MoveL RelTool (p1,3.000000,3.000000,9.000000,\Rx:=0.000000,\Ry:=0),vel1,zoneval,Extruder\WObj:=Workobject_1;
MoveL RelTool (p1,5.000000,3.000000,9.000000,\Rx:=0.000000,\Ry:=-0.000000),vel1,zoneval,Extruder\WObj:=Workobject_1;
MoveL RelTool (p1,7.500000,3.000000,9.000000,\Rx:=0.000000,\Ry:=-0.000000),vel1,zoneval,Extruder\WObj:=Workobject_1;
MoveL RelTool (p1,10.000000,3.000000,9.000000,\Rx:=0.000000,\Ry:=-0.000000),vel1,zoneval,Extruder\WObj:=Workobject_1;
MoveL RelTool (p1,12.500000,3.000000,9.000000,\Rx:=0.000000,\Ry:=-0.000000),vel1,zoneval,Extruder\WObj:=Workobject_1;
MoveL RelTool (p1,15.000000,3.000000,9.000000,\Rx:=0.000000,\Ry:=-0.000000),vel1,zoneval,Extruder\WObj:=Workobject_1;
MoveL RelTool (p1,17.500000,3.000000,9.083964,\Rx:=0.000000,\Ry:=-4.411855),vel1,zoneval,Extruder\WObj:=Workobject_1;
MoveL RelTool (p1,20.000000,3.000000,11.367111,\Rx:=0.000000,\Ry:=-10.154539),vel1,zoneval,Extruder\WObj:=Workobject_1;
MoveL RelTool (p1,22.500000,3.000000,13.528177,\Rx:=0.000000,\Ry:=-7.985654),vel1,zoneval,Extruder\WObj:=Workobject_1;
MoveL RelTool (p1,25.000000,3.000000,15.076143,\Rx:=0.000000,\Ry:=-5.751524),vel1,zoneval,Extruder\WObj:=Workobject_1;
MoveL RelTool (p1,27.500000,3.000000,16.224522,\Rx:=0.000000,\Ry:=-4.442626),vel1,zoneval,Extruder\WObj:=Workobject_1;
MoveL RelTool (p1,30.000000,3.000000,17.115741,\Rx:=0.000000,\Ry:=-3.471339),vel1,zoneval,Extruder\WObj:=Workobject_1;
MoveL RelTool (p1,32.500000,3.000000,17.811501,\Rx:=0.000000,\Ry:=-2.537038),vel1,zoneval,Extruder\WObj:=Workobject_1;
MoveL RelTool (p1,35.000000,3.000000,18.316346,\Rx:=0.000000,\Ry:=-2.278631),vel1,zoneval,Extruder\WObj:=Workobject_1;
MoveL RelTool (p1,37.500000,3.000000,18.667838,\Rx:=0.000000,\Ry:=-1.652509),vel1,zoneval,Extruder\WObj:=Workobject_1;
MoveL RelTool (p1,40.000000,3.000000,18.885153,\Rx:=0.000000,\Ry:=-0.809967),vel1,zoneval,Extruder\WObj:=Workobject_1;
MoveL RelTool (p1,42.500000,3.000000,18.988071,\Rx:=0.000000,\Ry:=-0.131676),vel1,zoneval,Extruder\WObj:=Workobject_1;
MoveL RelTool (p1,45.000000,3.000000,18.928943,\Rx:=0.000000,\Ry:=0.547333),vel1,zoneval,Extruder\WObj:=Workobject_1;
MoveL RelTool (p1,47.500000,3.000000,18.755880,\Rx:=0.000000,\Ry:=1.375675),vel1,zoneval,Extruder\WObj:=Workobject_1;
MoveL RelTool (p1,50.000000,3.000000,18.449475,\Rx:=0.000000,\Ry:=2.217990),vel1,zoneval,Extruder\WObj:=Workobject_1;
MoveL RelTool (p1,52.500000,3.000000,17.996328,\Rx:=0.000000,\Ry:=3.108480),vel1,zoneval,Extruder\WObj:=Workobject_1;
MoveL RelTool (p1,55.000000,3.000000,17.373557,\Rx:=0.000000,\Ry:=4.006255),vel1,zoneval,Extruder\WObj:=Workobject_1;
MoveL RelTool (p1,57.500000,3.000000,16.553376,\Rx:=0.000000,\Ry:=5.005887),vel1,zoneval,Extruder\WObj:=Workobject_1;
MoveL RelTool (p1,60.000000,3.000000,15.484711,\Rx:=0.000000,\Ry:=6.061214),vel1,zoneval,Extruder\WObj:=Workobject_1;
MoveL RelTool (p1,62.500000,3.000000,14.090610,\Rx:=0.000000,\Ry:=7.227695),vel1,zoneval,Extruder\WObj:=Workobject_1;
MoveL RelTool (p1,65.000000,3.000000,12.198583,\Rx:=0.000000,\Ry:=9.902860),vel1,zoneval,Extruder\WObj:=Workobject_1;
MoveL RelTool (p1,67.500000,3.000000,9.464073,\Rx:=0.000000,\Ry:=6.326197),vel1,zoneval,Extruder\WObj:=Workobject_1;
MoveL RelTool (p1,70.000000,3.000000,9.000000,\Rx:=0.000000,\Ry:=-0.000000),vel1,zoneval,Extruder\WObj:=Workobject_1;
MoveL RelTool (p1,72.500000,3.000000,9.000000,\Rx:=0.000000,\Ry:=-0.000000),vel1,zoneval,Extruder\WObj:=Workobject_1;
MoveL RelTool (p1,75.000000,3.000000,9.000000,\Rx:=0.000000,\Ry:=-0.000000),vel1,zoneval,Extruder\WObj:=Workobject_1;
MoveL RelTool (p1,77.500000,3.000000,9.000000,\Rx:=0.000000,\Ry:=-0.000000),vel1,zoneval,Extruder\WObj:=Workobject_1;
MoveL RelTool (p1,80.000000,3.000000,9.000000,\Rx:=0.000000,\Ry:=-0.000000),vel1,zoneval,Extruder\WObj:=Workobject_1;
MoveL RelTool (p1,82.500000,3.000000,9.000000,\Rx:=0.000000,\Ry:=-0.000000),vel1,zoneval,Extruder\WObj:=Workobject_1;
MoveL RelTool (p1,80.500000,3.500000,9.000000,\Rx:=0.000000,\Ry:=0.000000),vel1,zoneval,Extruder\WObj:=Workobject_1;
MoveL RelTool (p1,78.000000,3.500000,9.000000,\Rx:=0.000000,\Ry:=0.000000),vel1,zoneval,Extruder\WObj:=Workobject_1;
MoveL RelTool (p1,75.500000,3.500000,9.000000,\Rx:=0.000000,\Ry:=0.000000),vel1,zoneval,Extruder\WObj:=Workobject_1;
MoveL RelTool (p1,73.000000,3.500000,9.000000,\Rx:=0.000000,\Ry:=0.000000),vel1,zoneval,Extruder\WObj:=Workobject_1;
MoveL RelTool (p1,70.500000,3.500000,9.000000,\Rx:=0.000000,\Ry:=0.000000),vel1,zoneval,Extruder\WObj:=Workobject_1;
MoveL RelTool (p1,68.000000,3.500000,9.192958,\Rx:=0.000000,\Ry:=6.326197),vel1,zoneval,Extruder\WObj:=Workobject_1;
MoveL RelTool (p1,65.500000,3.500000,11.706154,\Rx:=0.000000,\Ry:=9.902860),vel1,zoneval,Extruder\WObj:=Workobject_1;
MoveL RelTool (p1,63.000000,3.500000,13.771773,\Rx:=0.000000,\Ry:=7.227695),vel1,zoneval,Extruder\WObj:=Workobject_1;
MoveL RelTool (p1,60.500000,3.500000,15.226913,\Rx:=0.000000,\Ry:=6.061214),vel1,zoneval,Extruder\WObj:=Workobject_1;
MoveL RelTool (p1,58.000000,3.500000,16.345998,\Rx:=0.000000,\Ry:=5.005887),vel1,zoneval,Extruder\WObj:=Workobject_1;
MoveL RelTool (p1,55.500000,3.500000,17.210825,\Rx:=0.000000,\Ry:=4.006255),vel1,zoneval,Extruder\WObj:=Workobject_1;
MoveL RelTool (p1,53.000000,3.500000,17.871774,\Rx:=0.000000,\Ry:=3.108480),vel1,zoneval,Extruder\WObj:=Workobject_1;
MoveL RelTool (p1,50.500000,3.500000,18.361483,\Rx:=0.000000,\Ry:=2.217990),vel1,zoneval,Extruder\WObj:=Workobject_1;
MoveL RelTool (p1,48.000000,3.500000,18.701647,\Rx:=0.000000,\Ry:=1.375675),vel1,zoneval,Extruder\WObj:=Workobject_1;
MoveL RelTool (p1,45.500000,3.500000,18.907436,\Rx:=0.000000,\Ry:=0.547333),vel1,zoneval,Extruder\WObj:=Workobject_1;
MoveL RelTool (p1,43.000000,3.500000,18.993242,\Rx:=0.000000,\Ry:=-0.131676),vel1,zoneval,Extruder\WObj:=Workobject_1;
MoveL RelTool (p1,40.500000,3.500000,18.917003,\Rx:=0.000000,\Ry:=-0.809967),vel1,zoneval,Extruder\WObj:=Workobject_1;
MoveL RelTool (p1,38.000000,3.500000,18.733099,\Rx:=0.000000,\Ry:=-1.652509),vel1,zoneval,Extruder\WObj:=Workobject_1;
MoveL RelTool (p1,35.500000,3.500000,18.406795,\Rx:=0.000000,\Ry:=-2.278631),vel1,zoneval,Extruder\WObj:=Workobject_1;
MoveL RelTool (p1,33.000000,3.500000,17.912470,\Rx:=0.000000,\Ry:=-2.537038),vel1,zoneval,Extruder\WObj:=Workobject_1;
MoveL RelTool (p1,30.500000,3.500000,17.255542,\Rx:=0.000000,\Ry:=-3.471339),vel1,zoneval,Extruder\WObj:=Workobject_1;
MoveL RelTool (p1,28.000000,3.500000,16.406426,\Rx:=0.000000,\Ry:=-4.442626),vel1,zoneval,Extruder\WObj:=Workobject_1;
MoveL RelTool (p1,25.500000,3.500000,15.318735,\Rx:=0.000000,\Ry:=-5.751524),vel1,zoneval,Extruder\WObj:=Workobject_1;
MoveL RelTool (p1,23.000000,3.500000,13.890588,\Rx:=0.000000,\Ry:=-7.985654),vel1,zoneval,Extruder\WObj:=Workobject_1;
MoveL RelTool (p1,20.500000,3.500000,11.879398,\Rx:=0.000000,\Ry:=-10.154539),vel1,zoneval,Extruder\WObj:=Workobject_1;
MoveL RelTool (p1,18.000000,3.500000,9.264501,\Rx:=0.000000,\Ry:=-4.411855),vel1,zoneval,Extruder\WObj:=Workobject_1;
MoveL RelTool (p1,15.500000,3.500000,9.000000,\Rx:=0.000000,\Ry:=0.000000),vel1,zoneval,Extruder\WObj:=Workobject_1;
MoveL RelTool (p1,13.000000,3.500000,9.000000,\Rx:=0.000000,\Ry:=0.000000),vel1,zoneval,Extruder\WObj:=Workobject_1;
MoveL RelTool (p1,10.500000,3.500000,9.000000,\Rx:=0.000000,\Ry:=0.000000),vel1,zoneval,Extruder\WObj:=Workobject_1;
MoveL RelTool (p1,8.000000,3.500000,9.000000,\Rx:=0.000000,\Ry:=0.000000),vel1,zoneval,Extruder\WObj:=Workobject_1;
MoveL RelTool (p1,5.500000,3.500000,9.000000,\Rx:=0.000000,\Ry:=0.000000),vel1,zoneval,Extruder\WObj:=Workobject_1;
MoveL RelTool (p1,3.000000,3.500000,9.000000,\Rx:=0.000000,\Ry:=0.000000),vel1,zoneval,Extruder\WObj:=Workobject_1;
MoveL RelTool (p1,5.000000,4.000000,9.000000,\Rx:=0.000000,\Ry:=-0.000000),vel1,zoneval,Extruder\WObj:=Workobject_1;
MoveL RelTool (p1,7.500000,4.000000,9.000000,\Rx:=0.000000,\Ry:=-0.000000),vel1,zoneval,Extruder\WObj:=Workobject_1;
MoveL RelTool (p1,10.000000,4.000000,9.000000,\Rx:=0.000000,\Ry:=-0.000000),vel1,zoneval,Extruder\WObj:=Workobject_1;
MoveL RelTool (p1,12.500000,4.000000,9.000000,\Rx:=0.000000,\Ry:=-0.000000),vel1,zoneval,Extruder\WObj:=Workobject_1;
MoveL RelTool (p1,15.000000,4.000000,9.000000,\Rx:=0.000000,\Ry:=-0.000000),vel1,zoneval,Extruder\WObj:=Workobject_1;
MoveL RelTool (p1,17.500000,4.000000,9.083964,\Rx:=0.000000,\Ry:=-4.411855),vel1,zoneval,Extruder\WObj:=Workobject_1;
MoveL RelTool (p1,20.000000,4.000000,11.367111,\Rx:=0.000000,\Ry:=-10.154539),vel1,zoneval,Extruder\WObj:=Workobject_1;
MoveL RelTool (p1,22.500000,4.000000,13.528177,\Rx:=0.000000,\Ry:=-7.985654),vel1,zoneval,Extruder\WObj:=Workobject_1;
MoveL RelTool (p1,25.000000,4.000000,15.076143,\Rx:=0.000000,\Ry:=-5.751524),vel1,zoneval,Extruder\WObj:=Workobject_1;
MoveL RelTool (p1,27.500000,4.000000,16.224522,\Rx:=0.000000,\Ry:=-4.442626),vel1,zoneval,Extruder\WObj:=Workobject_1;
MoveL RelTool (p1,30.000000,4.000000,17.115741,\Rx:=0.000000,\Ry:=-3.471339),vel1,zoneval,Extruder\WObj:=Workobject_1;
MoveL RelTool (p1,32.500000,4.000000,17.811501,\Rx:=0.000000,\Ry:=-2.537038),vel1,zoneval,Extruder\WObj:=Workobject_1;
MoveL RelTool (p1,35.000000,4.000000,18.316346,\Rx:=0.000000,\Ry:=-2.278631),vel1,zoneval,Extruder\WObj:=Workobject_1;
MoveL RelTool (p1,37.500000,4.000000,18.667838,\Rx:=0.000000,\Ry:=-1.652509),vel1,zoneval,Extruder\WObj:=Workobject_1;
MoveL RelTool (p1,40.000000,4.000000,18.885153,\Rx:=0.000000,\Ry:=-0.809967),vel1,zoneval,Extruder\WObj:=Workobject_1;
MoveL RelTool (p1,42.500000,4.000000,18.988071,\Rx:=0.000000,\Ry:=-0.131676),vel1,zoneval,Extruder\WObj:=Workobject_1;
MoveL RelTool (p1,45.000000,4.000000,18.928943,\Rx:=0.000000,\Ry:=0.547333),vel1,zoneval,Extruder\WObj:=Workobject_1;
MoveL RelTool (p1,47.500000,4.000000,18.755880,\Rx:=0.000000,\Ry:=1.375675),vel1,zoneval,Extruder\WObj:=Workobject_1;
MoveL RelTool (p1,50.000000,4.000000,18.449475,\Rx:=0.000000,\Ry:=2.217990),vel1,zoneval,Extruder\WObj:=Workobject_1;
MoveL RelTool (p1,52.500000,4.000000,17.996328,\Rx:=0.000000,\Ry:=3.108480),vel1,zoneval,Extruder\WObj:=Workobject_1;
MoveL RelTool (p1,55.000000,4.000000,17.373557,\Rx:=0.000000,\Ry:=4.006255),vel1,zoneval,Extruder\WObj:=Workobject_1;
MoveL RelTool (p1,57.500000,4.000000,16.553376,\Rx:=0.000000,\Ry:=5.005887),vel1,zoneval,Extruder\WObj:=Workobject_1;
MoveL RelTool (p1,60.000000,4.000000,15.484711,\Rx:=0.000000,\Ry:=6.061214),vel1,zoneval,Extruder\WObj:=Workobject_1;
MoveL RelTool (p1,62.500000,4.000000,14.090610,\Rx:=0.000000,\Ry:=7.227695),vel1,zoneval,Extruder\WObj:=Workobject_1;
MoveL RelTool (p1,65.000000,4.000000,12.198583,\Rx:=0.000000,\Ry:=9.902860),vel1,zoneval,Extruder\WObj:=Workobject_1;
MoveL RelTool (p1,67.500000,4.000000,9.464073,\Rx:=0.000000,\Ry:=6.326197),vel1,zoneval,Extruder\WObj:=Workobject_1;
MoveL RelTool (p1,70.000000,4.000000,9.000000,\Rx:=0.000000,\Ry:=-0.000000),vel1,zoneval,Extruder\WObj:=Workobject_1;
MoveL RelTool (p1,72.500000,4.000000,9.000000,\Rx:=0.000000,\Ry:=-0.000000),vel1,zoneval,Extruder\WObj:=Workobject_1;
MoveL RelTool (p1,75.000000,4.000000,9.000000,\Rx:=0.000000,\Ry:=-0.000000),vel1,zoneval,Extruder\WObj:=Workobject_1;
MoveL RelTool (p1,77.500000,4.000000,9.000000,\Rx:=0.000000,\Ry:=-0.000000),vel1,zoneval,Extruder\WObj:=Workobject_1;
MoveL RelTool (p1,80.000000,4.000000,9.000000,\Rx:=0.000000,\Ry:=-0.000000),vel1,zoneval,Extruder\WObj:=Workobject_1;
MoveL RelTool (p1,82.500000,4.000000,9.000000,\Rx:=0.000000,\Ry:=-0.000000),vel1,zoneval,Extruder\WObj:=Workobject_1;
MoveL RelTool (p1,80.500000,4.500000,9.000000,\Rx:=0.000000,\Ry:=0.000000),vel1,zoneval,Extruder\WObj:=Workobject_1;
MoveL RelTool (p1,78.000000,4.500000,9.000000,\Rx:=0.000000,\Ry:=0.000000),vel1,zoneval,Extruder\WObj:=Workobject_1;
MoveL RelTool (p1,75.500000,4.500000,9.000000,\Rx:=0.000000,\Ry:=0.000000),vel1,zoneval,Extruder\WObj:=Workobject_1;
MoveL RelTool (p1,73.000000,4.500000,9.000000,\Rx:=0.000000,\Ry:=0.000000),vel1,zoneval,Extruder\WObj:=Workobject_1;
MoveL RelTool (p1,70.500000,4.500000,9.000000,\Rx:=0.000000,\Ry:=0.000000),vel1,zoneval,Extruder\WObj:=Workobject_1;
MoveL RelTool (p1,68.000000,4.500000,9.192958,\Rx:=0.000000,\Ry:=6.326197),vel1,zoneval,Extruder\WObj:=Workobject_1;
MoveL RelTool (p1,65.500000,4.500000,11.706154,\Rx:=0.000000,\Ry:=9.902860),vel1,zoneval,Extruder\WObj:=Workobject_1;
MoveL RelTool (p1,63.000000,4.500000,13.771773,\Rx:=0.000000,\Ry:=7.227695),vel1,zoneval,Extruder\WObj:=Workobject_1;
MoveL RelTool (p1,60.500000,4.500000,15.226913,\Rx:=0.000000,\Ry:=6.061214),vel1,zoneval,Extruder\WObj:=Workobject_1;
MoveL RelTool (p1,58.000000,4.500000,16.345998,\Rx:=0.000000,\Ry:=5.005887),vel1,zoneval,Extruder\WObj:=Workobject_1;
MoveL RelTool (p1,55.500000,4.500000,17.210825,\Rx:=0.000000,\Ry:=4.006255),vel1,zoneval,Extruder\WObj:=Workobject_1;
MoveL RelTool (p1,53.000000,4.500000,17.871774,\Rx:=0.000000,\Ry:=3.108480),vel1,zoneval,Extruder\WObj:=Workobject_1;
MoveL RelTool (p1,50.500000,4.500000,18.361483,\Rx:=0.000000,\Ry:=2.217990),vel1,zoneval,Extruder\WObj:=Workobject_1;
MoveL RelTool (p1,48.000000,4.500000,18.701647,\Rx:=0.000000,\Ry:=1.375675),vel1,zoneval,Extruder\WObj:=Workobject_1;
MoveL RelTool (p1,45.500000,4.500000,18.907436,\Rx:=0.000000,\Ry:=0.547333),vel1,zoneval,Extruder\WObj:=Workobject_1;
MoveL RelTool (p1,43.000000,4.500000,18.993242,\Rx:=0.000000,\Ry:=-0.131676),vel1,zoneval,Extruder\WObj:=Workobject_1;
MoveL RelTool (p1,40.500000,4.500000,18.917003,\Rx:=0.000000,\Ry:=-0.809967),vel1,zoneval,Extruder\WObj:=Workobject_1;
MoveL RelTool (p1,38.000000,4.500000,18.733099,\Rx:=0.000000,\Ry:=-1.652509),vel1,zoneval,Extruder\WObj:=Workobject_1;
MoveL RelTool (p1,35.500000,4.500000,18.406795,\Rx:=0.000000,\Ry:=-2.278631),vel1,zoneval,Extruder\WObj:=Workobject_1;
MoveL RelTool (p1,33.000000,4.500000,17.912470,\Rx:=0.000000,\Ry:=-2.537038),vel1,zoneval,Extruder\WObj:=Workobject_1;
MoveL RelTool (p1,30.500000,4.500000,17.255542,\Rx:=0.000000,\Ry:=-3.471339),vel1,zoneval,Extruder\WObj:=Workobject_1;
MoveL RelTool (p1,28.000000,4.500000,16.406426,\Rx:=0.000000,\Ry:=-4.442626),vel1,zoneval,Extruder\WObj:=Workobject_1;
MoveL RelTool (p1,25.500000,4.500000,15.318735,\Rx:=0.000000,\Ry:=-5.751524),vel1,zoneval,Extruder\WObj:=Workobject_1;
MoveL RelTool (p1,23.000000,4.500000,13.890588,\Rx:=0.000000,\Ry:=-7.985654),vel1,zoneval,Extruder\WObj:=Workobject_1;
MoveL RelTool (p1,20.500000,4.500000,11.879398,\Rx:=0.000000,\Ry:=-10.154539),vel1,zoneval,Extruder\WObj:=Workobject_1;
MoveL RelTool (p1,18.000000,4.500000,9.264501,\Rx:=0.000000,\Ry:=-4.411855),vel1,zoneval,Extruder\WObj:=Workobject_1;
MoveL RelTool (p1,15.500000,4.500000,9.000000,\Rx:=0.000000,\Ry:=0.000000),vel1,zoneval,Extruder\WObj:=Workobject_1;
MoveL RelTool (p1,13.000000,4.500000,9.000000,\Rx:=0.000000,\Ry:=0.000000),vel1,zoneval,Extruder\WObj:=Workobject_1;
MoveL RelTool (p1,10.500000,4.500000,9.000000,\Rx:=0.000000,\Ry:=0.000000),vel1,zoneval,Extruder\WObj:=Workobject_1;
MoveL RelTool (p1,8.000000,4.500000,9.000000,\Rx:=0.000000,\Ry:=0.000000),vel1,zoneval,Extruder\WObj:=Workobject_1;
MoveL RelTool (p1,5.500000,4.500000,9.000000,\Rx:=0.000000,\Ry:=0.000000),vel1,zoneval,Extruder\WObj:=Workobject_1;
MoveL RelTool (p1,3.000000,4.500000,9.000000,\Rx:=0.000000,\Ry:=0.000000),vel1,zoneval,Extruder\WObj:=Workobject_1;
MoveL RelTool (p1,5.000000,5.000000,9.000000,\Rx:=0.000000,\Ry:=-0.000000),vel1,zoneval,Extruder\WObj:=Workobject_1;
MoveL RelTool (p1,7.500000,5.000000,9.000000,\Rx:=0.000000,\Ry:=-0.000000),vel1,zoneval,Extruder\WObj:=Workobject_1;
MoveL RelTool (p1,10.000000,5.000000,9.000000,\Rx:=0.000000,\Ry:=-0.000000),vel1,zoneval,Extruder\WObj:=Workobject_1;
MoveL RelTool (p1,12.500000,5.000000,9.000000,\Rx:=0.000000,\Ry:=-0.000000),vel1,zoneval,Extruder\WObj:=Workobject_1;
MoveL RelTool (p1,15.000000,5.000000,9.000000,\Rx:=0.000000,\Ry:=-0.000000),vel1,zoneval,Extruder\WObj:=Workobject_1;
MoveL RelTool (p1,17.500000,5.000000,9.083964,\Rx:=0.000000,\Ry:=-4.411855),vel1,zoneval,Extruder\WObj:=Workobject_1;
MoveL RelTool (p1,20.000000,5.000000,11.367111,\Rx:=0.000000,\Ry:=-10.154539),vel1,zoneval,Extruder\WObj:=Workobject_1;
MoveL RelTool (p1,22.500000,5.000000,13.528177,\Rx:=0.000000,\Ry:=-7.985654),vel1,zoneval,Extruder\WObj:=Workobject_1;
MoveL RelTool (p1,25.000000,5.000000,15.076143,\Rx:=0.000000,\Ry:=-5.751524),vel1,zoneval,Extruder\WObj:=Workobject_1;
MoveL RelTool (p1,27.500000,5.000000,16.224522,\Rx:=0.000000,\Ry:=-4.442626),vel1,zoneval,Extruder\WObj:=Workobject_1;
MoveL RelTool (p1,30.000000,5.000000,17.115741,\Rx:=0.000000,\Ry:=-3.471339),vel1,zoneval,Extruder\WObj:=Workobject_1;
MoveL RelTool (p1,32.500000,5.000000,17.811501,\Rx:=0.000000,\Ry:=-2.537038),vel1,zoneval,Extruder\WObj:=Workobject_1;
MoveL RelTool (p1,35.000000,5.000000,18.316346,\Rx:=0.000000,\Ry:=-2.278631),vel1,zoneval,Extruder\WObj:=Workobject_1;
MoveL RelTool (p1,37.500000,5.000000,18.667838,\Rx:=0.000000,\Ry:=-1.652509),vel1,zoneval,Extruder\WObj:=Workobject_1;
MoveL RelTool (p1,40.000000,5.000000,18.885153,\Rx:=0.000000,\Ry:=-0.809967),vel1,zoneval,Extruder\WObj:=Workobject_1;
MoveL RelTool (p1,42.500000,5.000000,18.988071,\Rx:=0.000000,\Ry:=-0.131676),vel1,zoneval,Extruder\WObj:=Workobject_1;
MoveL RelTool (p1,45.000000,5.000000,18.928943,\Rx:=0.000000,\Ry:=0.547333),vel1,zoneval,Extruder\WObj:=Workobject_1;
MoveL RelTool (p1,47.500000,5.000000,18.755880,\Rx:=0.000000,\Ry:=1.375675),vel1,zoneval,Extruder\WObj:=Workobject_1;
MoveL RelTool (p1,50.000000,5.000000,18.449475,\Rx:=0.000000,\Ry:=2.217990),vel1,zoneval,Extruder\WObj:=Workobject_1;
MoveL RelTool (p1,52.500000,5.000000,17.996328,\Rx:=0.000000,\Ry:=3.108480),vel1,zoneval,Extruder\WObj:=Workobject_1;
MoveL RelTool (p1,55.000000,5.000000,17.373557,\Rx:=0.000000,\Ry:=4.006255),vel1,zoneval,Extruder\WObj:=Workobject_1;
MoveL RelTool (p1,57.500000,5.000000,16.553376,\Rx:=0.000000,\Ry:=5.005887),vel1,zoneval,Extruder\WObj:=Workobject_1;
MoveL RelTool (p1,60.000000,5.000000,15.484711,\Rx:=0.000000,\Ry:=6.061214),vel1,zoneval,Extruder\WObj:=Workobject_1;
MoveL RelTool (p1,62.500000,5.000000,14.090610,\Rx:=0.000000,\Ry:=7.227695),vel1,zoneval,Extruder\WObj:=Workobject_1;
MoveL RelTool (p1,65.000000,5.000000,12.198583,\Rx:=0.000000,\Ry:=9.902860),vel1,zoneval,Extruder\WObj:=Workobject_1;
MoveL RelTool (p1,67.500000,5.000000,9.464073,\Rx:=0.000000,\Ry:=6.326197),vel1,zoneval,Extruder\WObj:=Workobject_1;
MoveL RelTool (p1,70.000000,5.000000,9.000000,\Rx:=0.000000,\Ry:=-0.000000),vel1,zoneval,Extruder\WObj:=Workobject_1;
MoveL RelTool (p1,72.500000,5.000000,9.000000,\Rx:=0.000000,\Ry:=-0.000000),vel1,zoneval,Extruder\WObj:=Workobject_1;
MoveL RelTool (p1,75.000000,5.000000,9.000000,\Rx:=0.000000,\Ry:=-0.000000),vel1,zoneval,Extruder\WObj:=Workobject_1;
MoveL RelTool (p1,77.500000,5.000000,9.000000,\Rx:=0.000000,\Ry:=-0.000000),vel1,zoneval,Extruder\WObj:=Workobject_1;
MoveL RelTool (p1,80.000000,5.000000,9.000000,\Rx:=0.000000,\Ry:=-0.000000),vel1,zoneval,Extruder\WObj:=Workobject_1;
MoveL RelTool (p1,82.500000,5.000000,9.000000,\Rx:=0.000000,\Ry:=-0.000000),vel1,zoneval,Extruder\WObj:=Workobject_1;
MoveL RelTool (p1,80.500000,5.500000,9.000000,\Rx:=0.000000,\Ry:=0.000000),vel1,zoneval,Extruder\WObj:=Workobject_1;
MoveL RelTool (p1,78.000000,5.500000,9.000000,\Rx:=0.000000,\Ry:=0.000000),vel1,zoneval,Extruder\WObj:=Workobject_1;
MoveL RelTool (p1,75.500000,5.500000,9.000000,\Rx:=0.000000,\Ry:=0.000000),vel1,zoneval,Extruder\WObj:=Workobject_1;
MoveL RelTool (p1,73.000000,5.500000,9.000000,\Rx:=0.000000,\Ry:=0.000000),vel1,zoneval,Extruder\WObj:=Workobject_1;
MoveL RelTool (p1,70.500000,5.500000,9.000000,\Rx:=0.000000,\Ry:=0.000000),vel1,zoneval,Extruder\WObj:=Workobject_1;
MoveL RelTool (p1,68.000000,5.500000,9.192958,\Rx:=0.000000,\Ry:=6.326197),vel1,zoneval,Extruder\WObj:=Workobject_1;
MoveL RelTool (p1,65.500000,5.500000,11.706154,\Rx:=0.000000,\Ry:=9.902860),vel1,zoneval,Extruder\WObj:=Workobject_1;
MoveL RelTool (p1,63.000000,5.500000,13.771773,\Rx:=0.000000,\Ry:=7.227695),vel1,zoneval,Extruder\WObj:=Workobject_1;
MoveL RelTool (p1,60.500000,5.500000,15.226913,\Rx:=0.000000,\Ry:=6.061214),vel1,zoneval,Extruder\WObj:=Workobject_1;
MoveL RelTool (p1,58.000000,5.500000,16.345998,\Rx:=0.000000,\Ry:=5.005887),vel1,zoneval,Extruder\WObj:=Workobject_1;
MoveL RelTool (p1,55.500000,5.500000,17.210825,\Rx:=0.000000,\Ry:=4.006255),vel1,zoneval,Extruder\WObj:=Workobject_1;
MoveL RelTool (p1,53.000000,5.500000,17.871774,\Rx:=0.000000,\Ry:=3.108480),vel1,zoneval,Extruder\WObj:=Workobject_1;
MoveL RelTool (p1,50.500000,5.500000,18.361483,\Rx:=0.000000,\Ry:=2.217990),vel1,zoneval,Extruder\WObj:=Workobject_1;
MoveL RelTool (p1,48.000000,5.500000,18.701647,\Rx:=0.000000,\Ry:=1.375675),vel1,zoneval,Extruder\WObj:=Workobject_1;
MoveL RelTool (p1,45.500000,5.500000,18.907436,\Rx:=0.000000,\Ry:=0.547333),vel1,zoneval,Extruder\WObj:=Workobject_1;
MoveL RelTool (p1,43.000000,5.500000,18.993242,\Rx:=0.000000,\Ry:=-0.131676),vel1,zoneval,Extruder\WObj:=Workobject_1;
MoveL RelTool (p1,40.500000,5.500000,18.917003,\Rx:=0.000000,\Ry:=-0.809967),vel1,zoneval,Extruder\WObj:=Workobject_1;
MoveL RelTool (p1,38.000000,5.500000,18.733099,\Rx:=0.000000,\Ry:=-1.652509),vel1,zoneval,Extruder\WObj:=Workobject_1;
MoveL RelTool (p1,35.500000,5.500000,18.406795,\Rx:=0.000000,\Ry:=-2.278631),vel1,zoneval,Extruder\WObj:=Workobject_1;
MoveL RelTool (p1,33.000000,5.500000,17.912470,\Rx:=0.000000,\Ry:=-2.537038),vel1,zoneval,Extruder\WObj:=Workobject_1;
MoveL RelTool (p1,30.500000,5.500000,17.255542,\Rx:=0.000000,\Ry:=-3.471339),vel1,zoneval,Extruder\WObj:=Workobject_1;
MoveL RelTool (p1,28.000000,5.500000,16.406426,\Rx:=0.000000,\Ry:=-4.442626),vel1,zoneval,Extruder\WObj:=Workobject_1;
MoveL RelTool (p1,25.500000,5.500000,15.318735,\Rx:=0.000000,\Ry:=-5.751524),vel1,zoneval,Extruder\WObj:=Workobject_1;
MoveL RelTool (p1,23.000000,5.500000,13.890588,\Rx:=0.000000,\Ry:=-7.985654),vel1,zoneval,Extruder\WObj:=Workobject_1;
MoveL RelTool (p1,20.500000,5.500000,11.879398,\Rx:=0.000000,\Ry:=-10.154539),vel1,zoneval,Extruder\WObj:=Workobject_1;
MoveL RelTool (p1,18.000000,5.500000,9.264501,\Rx:=0.000000,\Ry:=-4.411855),vel1,zoneval,Extruder\WObj:=Workobject_1;
MoveL RelTool (p1,15.500000,5.500000,9.000000,\Rx:=0.000000,\Ry:=0.000000),vel1,zoneval,Extruder\WObj:=Workobject_1;
MoveL RelTool (p1,13.000000,5.500000,9.000000,\Rx:=0.000000,\Ry:=0.000000),vel1,zoneval,Extruder\WObj:=Workobject_1;
MoveL RelTool (p1,10.500000,5.500000,9.000000,\Rx:=0.000000,\Ry:=0.000000),vel1,zoneval,Extruder\WObj:=Workobject_1;
MoveL RelTool (p1,8.000000,5.500000,9.000000,\Rx:=0.000000,\Ry:=0.000000),vel1,zoneval,Extruder\WObj:=Workobject_1;
MoveL RelTool (p1,5.500000,5.500000,9.000000,\Rx:=0.000000,\Ry:=0.000000),vel1,zoneval,Extruder\WObj:=Workobject_1;
MoveL RelTool (p1,3.000000,5.500000,9.000000,\Rx:=0.000000,\Ry:=0.000000),vel1,zoneval,Extruder\WObj:=Workobject_1;
MoveL RelTool (p1,5.000000,6.000000,9.000000,\Rx:=0.000000,\Ry:=-0.000000),vel1,zoneval,Extruder\WObj:=Workobject_1;
MoveL RelTool (p1,7.500000,6.000000,9.000000,\Rx:=0.000000,\Ry:=-0.000000),vel1,zoneval,Extruder\WObj:=Workobject_1;
MoveL RelTool (p1,10.000000,6.000000,9.000000,\Rx:=0.000000,\Ry:=-0.000000),vel1,zoneval,Extruder\WObj:=Workobject_1;
MoveL RelTool (p1,12.500000,6.000000,9.000000,\Rx:=0.000000,\Ry:=-0.000000),vel1,zoneval,Extruder\WObj:=Workobject_1;
MoveL RelTool (p1,15.000000,6.000000,9.000000,\Rx:=0.000000,\Ry:=-0.000000),vel1,zoneval,Extruder\WObj:=Workobject_1;
MoveL RelTool (p1,17.500000,6.000000,9.083964,\Rx:=0.000000,\Ry:=-4.411855),vel1,zoneval,Extruder\WObj:=Workobject_1;
MoveL RelTool (p1,20.000000,6.000000,11.367111,\Rx:=0.000000,\Ry:=-10.154539),vel1,zoneval,Extruder\WObj:=Workobject_1;
MoveL RelTool (p1,22.500000,6.000000,13.528177,\Rx:=0.000000,\Ry:=-7.985654),vel1,zoneval,Extruder\WObj:=Workobject_1;
MoveL RelTool (p1,25.000000,6.000000,15.076143,\Rx:=0.000000,\Ry:=-5.751524),vel1,zoneval,Extruder\WObj:=Workobject_1;
MoveL RelTool (p1,27.500000,6.000000,16.224522,\Rx:=0.000000,\Ry:=-4.442626),vel1,zoneval,Extruder\WObj:=Workobject_1;
MoveL RelTool (p1,30.000000,6.000000,17.115741,\Rx:=0.000000,\Ry:=-3.471339),vel1,zoneval,Extruder\WObj:=Workobject_1;
MoveL RelTool (p1,32.500000,6.000000,17.811501,\Rx:=0.000000,\Ry:=-2.537038),vel1,zoneval,Extruder\WObj:=Workobject_1;
MoveL RelTool (p1,35.000000,6.000000,18.316346,\Rx:=0.000000,\Ry:=-2.278631),vel1,zoneval,Extruder\WObj:=Workobject_1;
MoveL RelTool (p1,37.500000,6.000000,18.667838,\Rx:=0.000000,\Ry:=-1.652509),vel1,zoneval,Extruder\WObj:=Workobject_1;
MoveL RelTool (p1,40.000000,6.000000,18.885153,\Rx:=0.000000,\Ry:=-0.809967),vel1,zoneval,Extruder\WObj:=Workobject_1;
MoveL RelTool (p1,42.500000,6.000000,18.988071,\Rx:=0.000000,\Ry:=-0.131676),vel1,zoneval,Extruder\WObj:=Workobject_1;
MoveL RelTool (p1,45.000000,6.000000,18.928943,\Rx:=0.000000,\Ry:=0.547333),vel1,zoneval,Extruder\WObj:=Workobject_1;
MoveL RelTool (p1,47.500000,6.000000,18.755880,\Rx:=0.000000,\Ry:=1.375675),vel1,zoneval,Extruder\WObj:=Workobject_1;
MoveL RelTool (p1,50.000000,6.000000,18.449475,\Rx:=0.000000,\Ry:=2.217990),vel1,zoneval,Extruder\WObj:=Workobject_1;
MoveL RelTool (p1,52.500000,6.000000,17.996328,\Rx:=0.000000,\Ry:=3.108480),vel1,zoneval,Extruder\WObj:=Workobject_1;
MoveL RelTool (p1,55.000000,6.000000,17.373557,\Rx:=0.000000,\Ry:=4.006255),vel1,zoneval,Extruder\WObj:=Workobject_1;
MoveL RelTool (p1,57.500000,6.000000,16.553376,\Rx:=0.000000,\Ry:=5.005887),vel1,zoneval,Extruder\WObj:=Workobject_1;
MoveL RelTool (p1,60.000000,6.000000,15.484711,\Rx:=0.000000,\Ry:=6.061214),vel1,zoneval,Extruder\WObj:=Workobject_1;
MoveL RelTool (p1,62.500000,6.000000,14.090610,\Rx:=0.000000,\Ry:=7.227695),vel1,zoneval,Extruder\WObj:=Workobject_1;
MoveL RelTool (p1,65.000000,6.000000,12.198583,\Rx:=0.000000,\Ry:=9.902860),vel1,zoneval,Extruder\WObj:=Workobject_1;
MoveL RelTool (p1,67.500000,6.000000,9.464073,\Rx:=0.000000,\Ry:=6.326197),vel1,zoneval,Extruder\WObj:=Workobject_1;
MoveL RelTool (p1,70.000000,6.000000,9.000000,\Rx:=0.000000,\Ry:=-0.000000),vel1,zoneval,Extruder\WObj:=Workobject_1;
MoveL RelTool (p1,72.500000,6.000000,9.000000,\Rx:=0.000000,\Ry:=-0.000000),vel1,zoneval,Extruder\WObj:=Workobject_1;
MoveL RelTool (p1,75.000000,6.000000,9.000000,\Rx:=0.000000,\Ry:=-0.000000),vel1,zoneval,Extruder\WObj:=Workobject_1;
MoveL RelTool (p1,77.500000,6.000000,9.000000,\Rx:=0.000000,\Ry:=-0.000000),vel1,zoneval,Extruder\WObj:=Workobject_1;
MoveL RelTool (p1,80.000000,6.000000,9.000000,\Rx:=0.000000,\Ry:=-0.000000),vel1,zoneval,Extruder\WObj:=Workobject_1;
MoveL RelTool (p1,82.500000,6.000000,9.000000,\Rx:=0.000000,\Ry:=-0.000000),vel1,zoneval,Extruder\WObj:=Workobject_1;
MoveL RelTool (p1,80.500000,6.500000,9.000000,\Rx:=0.000000,\Ry:=0.000000),vel1,zoneval,Extruder\WObj:=Workobject_1;
MoveL RelTool (p1,78.000000,6.500000,9.000000,\Rx:=0.000000,\Ry:=0.000000),vel1,zoneval,Extruder\WObj:=Workobject_1;
MoveL RelTool (p1,75.500000,6.500000,9.000000,\Rx:=0.000000,\Ry:=0.000000),vel1,zoneval,Extruder\WObj:=Workobject_1;
MoveL RelTool (p1,73.000000,6.500000,9.000000,\Rx:=0.000000,\Ry:=0.000000),vel1,zoneval,Extruder\WObj:=Workobject_1;
MoveL RelTool (p1,70.500000,6.500000,9.000000,\Rx:=0.000000,\Ry:=0.000000),vel1,zoneval,Extruder\WObj:=Workobject_1;
MoveL RelTool (p1,68.000000,6.500000,9.192958,\Rx:=0.000000,\Ry:=6.326197),vel1,zoneval,Extruder\WObj:=Workobject_1;
MoveL RelTool (p1,65.500000,6.500000,11.706154,\Rx:=0.000000,\Ry:=9.902860),vel1,zoneval,Extruder\WObj:=Workobject_1;
MoveL RelTool (p1,63.000000,6.500000,13.771773,\Rx:=0.000000,\Ry:=7.227695),vel1,zoneval,Extruder\WObj:=Workobject_1;
MoveL RelTool (p1,60.500000,6.500000,15.226913,\Rx:=0.000000,\Ry:=6.061214),vel1,zoneval,Extruder\WObj:=Workobject_1;
MoveL RelTool (p1,58.000000,6.500000,16.345998,\Rx:=0.000000,\Ry:=5.005887),vel1,zoneval,Extruder\WObj:=Workobject_1;
MoveL RelTool (p1,55.500000,6.500000,17.210825,\Rx:=0.000000,\Ry:=4.006255),vel1,zoneval,Extruder\WObj:=Workobject_1;
MoveL RelTool (p1,53.000000,6.500000,17.871774,\Rx:=0.000000,\Ry:=3.108480),vel1,zoneval,Extruder\WObj:=Workobject_1;
MoveL RelTool (p1,50.500000,6.500000,18.361483,\Rx:=0.000000,\Ry:=2.217990),vel1,zoneval,Extruder\WObj:=Workobject_1;
MoveL RelTool (p1,48.000000,6.500000,18.701647,\Rx:=0.000000,\Ry:=1.375675),vel1,zoneval,Extruder\WObj:=Workobject_1;
MoveL RelTool (p1,45.500000,6.500000,18.907436,\Rx:=0.000000,\Ry:=0.547333),vel1,zoneval,Extruder\WObj:=Workobject_1;
MoveL RelTool (p1,43.000000,6.500000,18.993242,\Rx:=0.000000,\Ry:=-0.131676),vel1,zoneval,Extruder\WObj:=Workobject_1;
MoveL RelTool (p1,40.500000,6.500000,18.917003,\Rx:=0.000000,\Ry:=-0.809967),vel1,zoneval,Extruder\WObj:=Workobject_1;
MoveL RelTool (p1,38.000000,6.500000,18.733099,\Rx:=0.000000,\Ry:=-1.652509),vel1,zoneval,Extruder\WObj:=Workobject_1;
MoveL RelTool (p1,35.500000,6.500000,18.406795,\Rx:=0.000000,\Ry:=-2.278631),vel1,zoneval,Extruder\WObj:=Workobject_1;
MoveL RelTool (p1,33.000000,6.500000,17.912470,\Rx:=0.000000,\Ry:=-2.537038),vel1,zoneval,Extruder\WObj:=Workobject_1;
MoveL RelTool (p1,30.500000,6.500000,17.255542,\Rx:=0.000000,\Ry:=-3.471339),vel1,zoneval,Extruder\WObj:=Workobject_1;
MoveL RelTool (p1,28.000000,6.500000,16.406426,\Rx:=0.000000,\Ry:=-4.442626),vel1,zoneval,Extruder\WObj:=Workobject_1;
MoveL RelTool (p1,25.500000,6.500000,15.318735,\Rx:=0.000000,\Ry:=-5.751524),vel1,zoneval,Extruder\WObj:=Workobject_1;
MoveL RelTool (p1,23.000000,6.500000,13.890588,\Rx:=0.000000,\Ry:=-7.985654),vel1,zoneval,Extruder\WObj:=Workobject_1;
MoveL RelTool (p1,20.500000,6.500000,11.879398,\Rx:=0.000000,\Ry:=-10.154539),vel1,zoneval,Extruder\WObj:=Workobject_1;
MoveL RelTool (p1,18.000000,6.500000,9.264501,\Rx:=0.000000,\Ry:=-4.411855),vel1,zoneval,Extruder\WObj:=Workobject_1;
MoveL RelTool (p1,15.500000,6.500000,9.000000,\Rx:=0.000000,\Ry:=0.000000),vel1,zoneval,Extruder\WObj:=Workobject_1;
MoveL RelTool (p1,13.000000,6.500000,9.000000,\Rx:=0.000000,\Ry:=0.000000),vel1,zoneval,Extruder\WObj:=Workobject_1;
MoveL RelTool (p1,10.500000,6.500000,9.000000,\Rx:=0.000000,\Ry:=0.000000),vel1,zoneval,Extruder\WObj:=Workobject_1;
MoveL RelTool (p1,8.000000,6.500000,9.000000,\Rx:=0.000000,\Ry:=0.000000),vel1,zoneval,Extruder\WObj:=Workobject_1;
MoveL RelTool (p1,5.500000,6.500000,9.000000,\Rx:=0.000000,\Ry:=0.000000),vel1,zoneval,Extruder\WObj:=Workobject_1;
MoveL RelTool (p1,3.000000,6.500000,9.000000,\Rx:=0.000000,\Ry:=0.000000),vel1,zoneval,Extruder\WObj:=Workobject_1;
MoveL RelTool (p1,5.000000,7.000000,9.000000,\Rx:=0.000000,\Ry:=-0.000000),vel1,zoneval,Extruder\WObj:=Workobject_1;
MoveL RelTool (p1,7.500000,7.000000,9.000000,\Rx:=0.000000,\Ry:=-0.000000),vel1,zoneval,Extruder\WObj:=Workobject_1;
MoveL RelTool (p1,10.000000,7.000000,9.000000,\Rx:=0.000000,\Ry:=-0.000000),vel1,zoneval,Extruder\WObj:=Workobject_1;
MoveL RelTool (p1,12.500000,7.000000,9.000000,\Rx:=0.000000,\Ry:=-0.000000),vel1,zoneval,Extruder\WObj:=Workobject_1;
MoveL RelTool (p1,15.000000,7.000000,9.000000,\Rx:=0.000000,\Ry:=-0.000000),vel1,zoneval,Extruder\WObj:=Workobject_1;
MoveL RelTool (p1,17.500000,7.000000,9.083964,\Rx:=0.000000,\Ry:=-4.411855),vel1,zoneval,Extruder\WObj:=Workobject_1;
MoveL RelTool (p1,20.000000,7.000000,11.367111,\Rx:=0.000000,\Ry:=-10.154539),vel1,zoneval,Extruder\WObj:=Workobject_1;
MoveL RelTool (p1,22.500000,7.000000,13.528177,\Rx:=0.000000,\Ry:=-7.985654),vel1,zoneval,Extruder\WObj:=Workobject_1;
MoveL RelTool (p1,25.000000,7.000000,15.076143,\Rx:=0.000000,\Ry:=-5.751524),vel1,zoneval,Extruder\WObj:=Workobject_1;
MoveL RelTool (p1,27.500000,7.000000,16.224522,\Rx:=0.000000,\Ry:=-4.442626),vel1,zoneval,Extruder\WObj:=Workobject_1;
MoveL RelTool (p1,30.000000,7.000000,17.115741,\Rx:=0.000000,\Ry:=-3.471339),vel1,zoneval,Extruder\WObj:=Workobject_1;
MoveL RelTool (p1,32.500000,7.000000,17.811501,\Rx:=0.000000,\Ry:=-2.537038),vel1,zoneval,Extruder\WObj:=Workobject_1;
MoveL RelTool (p1,35.000000,7.000000,18.316346,\Rx:=0.000000,\Ry:=-2.278631),vel1,zoneval,Extruder\WObj:=Workobject_1;
MoveL RelTool (p1,37.500000,7.000000,18.667838,\Rx:=0.000000,\Ry:=-1.652509),vel1,zoneval,Extruder\WObj:=Workobject_1;
MoveL RelTool (p1,40.000000,7.000000,18.885153,\Rx:=0.000000,\Ry:=-0.809967),vel1,zoneval,Extruder\WObj:=Workobject_1;
MoveL RelTool (p1,42.500000,7.000000,18.988071,\Rx:=0.000000,\Ry:=-0.131676),vel1,zoneval,Extruder\WObj:=Workobject_1;
MoveL RelTool (p1,45.000000,7.000000,18.928943,\Rx:=0.000000,\Ry:=0.547333),vel1,zoneval,Extruder\WObj:=Workobject_1;
MoveL RelTool (p1,47.500000,7.000000,18.755880,\Rx:=0.000000,\Ry:=1.375675),vel1,zoneval,Extruder\WObj:=Workobject_1;
MoveL RelTool (p1,50.000000,7.000000,18.449475,\Rx:=0.000000,\Ry:=2.217990),vel1,zoneval,Extruder\WObj:=Workobject_1;
MoveL RelTool (p1,52.500000,7.000000,17.996328,\Rx:=0.000000,\Ry:=3.108480),vel1,zoneval,Extruder\WObj:=Workobject_1;
MoveL RelTool (p1,55.000000,7.000000,17.373557,\Rx:=0.000000,\Ry:=4.006255),vel1,zoneval,Extruder\WObj:=Workobject_1;
MoveL RelTool (p1,57.500000,7.000000,16.553376,\Rx:=0.000000,\Ry:=5.005887),vel1,zoneval,Extruder\WObj:=Workobject_1;
MoveL RelTool (p1,60.000000,7.000000,15.484711,\Rx:=0.000000,\Ry:=6.061214),vel1,zoneval,Extruder\WObj:=Workobject_1;
MoveL RelTool (p1,62.500000,7.000000,14.090610,\Rx:=0.000000,\Ry:=7.227695),vel1,zoneval,Extruder\WObj:=Workobject_1;
MoveL RelTool (p1,65.000000,7.000000,12.198583,\Rx:=0.000000,\Ry:=9.902860),vel1,zoneval,Extruder\WObj:=Workobject_1;
MoveL RelTool (p1,67.500000,7.000000,9.464073,\Rx:=0.000000,\Ry:=6.326197),vel1,zoneval,Extruder\WObj:=Workobject_1;
MoveL RelTool (p1,70.000000,7.000000,9.000000,\Rx:=0.000000,\Ry:=-0.000000),vel1,zoneval,Extruder\WObj:=Workobject_1;
MoveL RelTool (p1,72.500000,7.000000,9.000000,\Rx:=0.000000,\Ry:=-0.000000),vel1,zoneval,Extruder\WObj:=Workobject_1;
MoveL RelTool (p1,75.000000,7.000000,9.000000,\Rx:=0.000000,\Ry:=-0.000000),vel1,zoneval,Extruder\WObj:=Workobject_1;
MoveL RelTool (p1,77.500000,7.000000,9.000000,\Rx:=0.000000,\Ry:=-0.000000),vel1,zoneval,Extruder\WObj:=Workobject_1;
MoveL RelTool (p1,80.000000,7.000000,9.000000,\Rx:=0.000000,\Ry:=-0.000000),vel1,zoneval,Extruder\WObj:=Workobject_1;
MoveL RelTool (p1,82.500000,7.000000,9.000000,\Rx:=0.000000,\Ry:=-0.000000),vel1,zoneval,Extruder\WObj:=Workobject_1;
MoveL RelTool (p1,80.500000,7.500000,9.000000,\Rx:=0.000000,\Ry:=0.000000),vel1,zoneval,Extruder\WObj:=Workobject_1;
MoveL RelTool (p1,78.000000,7.500000,9.000000,\Rx:=0.000000,\Ry:=0.000000),vel1,zoneval,Extruder\WObj:=Workobject_1;
MoveL RelTool (p1,75.500000,7.500000,9.000000,\Rx:=0.000000,\Ry:=0.000000),vel1,zoneval,Extruder\WObj:=Workobject_1;
MoveL RelTool (p1,73.000000,7.500000,9.000000,\Rx:=0.000000,\Ry:=0.000000),vel1,zoneval,Extruder\WObj:=Workobject_1;
MoveL RelTool (p1,70.500000,7.500000,9.000000,\Rx:=0.000000,\Ry:=0.000000),vel1,zoneval,Extruder\WObj:=Workobject_1;
MoveL RelTool (p1,68.000000,7.500000,9.192958,\Rx:=0.000000,\Ry:=6.326197),vel1,zoneval,Extruder\WObj:=Workobject_1;
MoveL RelTool (p1,65.500000,7.500000,11.706154,\Rx:=0.000000,\Ry:=9.902860),vel1,zoneval,Extruder\WObj:=Workobject_1;
MoveL RelTool (p1,63.000000,7.500000,13.771773,\Rx:=0.000000,\Ry:=7.227695),vel1,zoneval,Extruder\WObj:=Workobject_1;
MoveL RelTool (p1,60.500000,7.500000,15.226913,\Rx:=0.000000,\Ry:=6.061214),vel1,zoneval,Extruder\WObj:=Workobject_1;
MoveL RelTool (p1,58.000000,7.500000,16.345998,\Rx:=0.000000,\Ry:=5.005887),vel1,zoneval,Extruder\WObj:=Workobject_1;
MoveL RelTool (p1,55.500000,7.500000,17.210825,\Rx:=0.000000,\Ry:=4.006255),vel1,zoneval,Extruder\WObj:=Workobject_1;
MoveL RelTool (p1,53.000000,7.500000,17.871774,\Rx:=0.000000,\Ry:=3.108480),vel1,zoneval,Extruder\WObj:=Workobject_1;
MoveL RelTool (p1,50.500000,7.500000,18.361483,\Rx:=0.000000,\Ry:=2.217990),vel1,zoneval,Extruder\WObj:=Workobject_1;
MoveL RelTool (p1,48.000000,7.500000,18.701647,\Rx:=0.000000,\Ry:=1.375675),vel1,zoneval,Extruder\WObj:=Workobject_1;
MoveL RelTool (p1,45.500000,7.500000,18.907436,\Rx:=0.000000,\Ry:=0.547333),vel1,zoneval,Extruder\WObj:=Workobject_1;
MoveL RelTool (p1,43.000000,7.500000,18.993242,\Rx:=0.000000,\Ry:=-0.131676),vel1,zoneval,Extruder\WObj:=Workobject_1;
MoveL RelTool (p1,40.500000,7.500000,18.917003,\Rx:=0.000000,\Ry:=-0.809967),vel1,zoneval,Extruder\WObj:=Workobject_1;
MoveL RelTool (p1,38.000000,7.500000,18.733099,\Rx:=0.000000,\Ry:=-1.652509),vel1,zoneval,Extruder\WObj:=Workobject_1;
MoveL RelTool (p1,35.500000,7.500000,18.406795,\Rx:=0.000000,\Ry:=-2.278631),vel1,zoneval,Extruder\WObj:=Workobject_1;
MoveL RelTool (p1,33.000000,7.500000,17.912470,\Rx:=0.000000,\Ry:=-2.537038),vel1,zoneval,Extruder\WObj:=Workobject_1;
MoveL RelTool (p1,30.500000,7.500000,17.255542,\Rx:=0.000000,\Ry:=-3.471339),vel1,zoneval,Extruder\WObj:=Workobject_1;
MoveL RelTool (p1,28.000000,7.500000,16.406426,\Rx:=0.000000,\Ry:=-4.442626),vel1,zoneval,Extruder\WObj:=Workobject_1;
MoveL RelTool (p1,25.500000,7.500000,15.318735,\Rx:=0.000000,\Ry:=-5.751524),vel1,zoneval,Extruder\WObj:=Workobject_1;
MoveL RelTool (p1,23.000000,7.500000,13.890588,\Rx:=0.000000,\Ry:=-7.985654),vel1,zoneval,Extruder\WObj:=Workobject_1;
MoveL RelTool (p1,20.500000,7.500000,11.879398,\Rx:=0.000000,\Ry:=-10.154539),vel1,zoneval,Extruder\WObj:=Workobject_1;
MoveL RelTool (p1,18.000000,7.500000,9.264501,\Rx:=0.000000,\Ry:=-4.411855),vel1,zoneval,Extruder\WObj:=Workobject_1;
MoveL RelTool (p1,15.500000,7.500000,9.000000,\Rx:=0.000000,\Ry:=0.000000),vel1,zoneval,Extruder\WObj:=Workobject_1;
MoveL RelTool (p1,13.000000,7.500000,9.000000,\Rx:=0.000000,\Ry:=0.000000),vel1,zoneval,Extruder\WObj:=Workobject_1;
MoveL RelTool (p1,10.500000,7.500000,9.000000,\Rx:=0.000000,\Ry:=0.000000),vel1,zoneval,Extruder\WObj:=Workobject_1;
MoveL RelTool (p1,8.000000,7.500000,9.000000,\Rx:=0.000000,\Ry:=0.000000),vel1,zoneval,Extruder\WObj:=Workobject_1;
MoveL RelTool (p1,5.500000,7.500000,9.000000,\Rx:=0.000000,\Ry:=0.000000),vel1,zoneval,Extruder\WObj:=Workobject_1;
MoveL RelTool (p1,3.000000,7.500000,9.000000,\Rx:=0.000000,\Ry:=0.000000),vel1,zoneval,Extruder\WObj:=Workobject_1;
MoveL RelTool (p1,5.000000,8.000000,9.000000,\Rx:=0.000000,\Ry:=-0.000000),vel1,zoneval,Extruder\WObj:=Workobject_1;
MoveL RelTool (p1,7.500000,8.000000,9.000000,\Rx:=0.000000,\Ry:=-0.000000),vel1,zoneval,Extruder\WObj:=Workobject_1;
MoveL RelTool (p1,10.000000,8.000000,9.000000,\Rx:=0.000000,\Ry:=-0.000000),vel1,zoneval,Extruder\WObj:=Workobject_1;
MoveL RelTool (p1,12.500000,8.000000,9.000000,\Rx:=0.000000,\Ry:=-0.000000),vel1,zoneval,Extruder\WObj:=Workobject_1;
MoveL RelTool (p1,15.000000,8.000000,9.000000,\Rx:=0.000000,\Ry:=-0.000000),vel1,zoneval,Extruder\WObj:=Workobject_1;
MoveL RelTool (p1,17.500000,8.000000,9.083964,\Rx:=0.000000,\Ry:=-4.411855),vel1,zoneval,Extruder\WObj:=Workobject_1;
MoveL RelTool (p1,20.000000,8.000000,11.367111,\Rx:=0.000000,\Ry:=-10.154539),vel1,zoneval,Extruder\WObj:=Workobject_1;
MoveL RelTool (p1,22.500000,8.000000,13.528177,\Rx:=0.000000,\Ry:=-7.985654),vel1,zoneval,Extruder\WObj:=Workobject_1;
MoveL RelTool (p1,25.000000,8.000000,15.076143,\Rx:=0.000000,\Ry:=-5.751524),vel1,zoneval,Extruder\WObj:=Workobject_1;
MoveL RelTool (p1,27.500000,8.000000,16.224522,\Rx:=0.000000,\Ry:=-4.442626),vel1,zoneval,Extruder\WObj:=Workobject_1;
MoveL RelTool (p1,30.000000,8.000000,17.115741,\Rx:=0.000000,\Ry:=-3.471339),vel1,zoneval,Extruder\WObj:=Workobject_1;
MoveL RelTool (p1,32.500000,8.000000,17.811501,\Rx:=0.000000,\Ry:=-2.537038),vel1,zoneval,Extruder\WObj:=Workobject_1;
MoveL RelTool (p1,35.000000,8.000000,18.316346,\Rx:=0.000000,\Ry:=-2.278631),vel1,zoneval,Extruder\WObj:=Workobject_1;
MoveL RelTool (p1,37.500000,8.000000,18.667838,\Rx:=0.000000,\Ry:=-1.652509),vel1,zoneval,Extruder\WObj:=Workobject_1;
MoveL RelTool (p1,40.000000,8.000000,18.885153,\Rx:=0.000000,\Ry:=-0.809967),vel1,zoneval,Extruder\WObj:=Workobject_1;
MoveL RelTool (p1,42.500000,8.000000,18.988071,\Rx:=0.000000,\Ry:=-0.131676),vel1,zoneval,Extruder\WObj:=Workobject_1;
MoveL RelTool (p1,45.000000,8.000000,18.928943,\Rx:=0.000000,\Ry:=0.547333),vel1,zoneval,Extruder\WObj:=Workobject_1;
MoveL RelTool (p1,47.500000,8.000000,18.755880,\Rx:=0.000000,\Ry:=1.375675),vel1,zoneval,Extruder\WObj:=Workobject_1;
MoveL RelTool (p1,50.000000,8.000000,18.449475,\Rx:=0.000000,\Ry:=2.217990),vel1,zoneval,Extruder\WObj:=Workobject_1;
MoveL RelTool (p1,52.500000,8.000000,17.996328,\Rx:=0.000000,\Ry:=3.108480),vel1,zoneval,Extruder\WObj:=Workobject_1;
MoveL RelTool (p1,55.000000,8.000000,17.373557,\Rx:=0.000000,\Ry:=4.006255),vel1,zoneval,Extruder\WObj:=Workobject_1;
MoveL RelTool (p1,57.500000,8.000000,16.553376,\Rx:=0.000000,\Ry:=5.005887),vel1,zoneval,Extruder\WObj:=Workobject_1;
MoveL RelTool (p1,60.000000,8.000000,15.484711,\Rx:=0.000000,\Ry:=6.061214),vel1,zoneval,Extruder\WObj:=Workobject_1;
MoveL RelTool (p1,62.500000,8.000000,14.090610,\Rx:=0.000000,\Ry:=7.227695),vel1,zoneval,Extruder\WObj:=Workobject_1;
MoveL RelTool (p1,65.000000,8.000000,12.198583,\Rx:=0.000000,\Ry:=9.902860),vel1,zoneval,Extruder\WObj:=Workobject_1;
MoveL RelTool (p1,67.500000,8.000000,9.464073,\Rx:=0.000000,\Ry:=6.326197),vel1,zoneval,Extruder\WObj:=Workobject_1;
MoveL RelTool (p1,70.000000,8.000000,9.000000,\Rx:=0.000000,\Ry:=-0.000000),vel1,zoneval,Extruder\WObj:=Workobject_1;
MoveL RelTool (p1,72.500000,8.000000,9.000000,\Rx:=0.000000,\Ry:=-0.000000),vel1,zoneval,Extruder\WObj:=Workobject_1;
MoveL RelTool (p1,75.000000,8.000000,9.000000,\Rx:=0.000000,\Ry:=-0.000000),vel1,zoneval,Extruder\WObj:=Workobject_1;
MoveL RelTool (p1,77.500000,8.000000,9.000000,\Rx:=0.000000,\Ry:=-0.000000),vel1,zoneval,Extruder\WObj:=Workobject_1;
MoveL RelTool (p1,80.000000,8.000000,9.000000,\Rx:=0.000000,\Ry:=-0.000000),vel1,zoneval,Extruder\WObj:=Workobject_1;
MoveL RelTool (p1,82.500000,8.000000,9.000000,\Rx:=0.000000,\Ry:=-0.000000),vel1,zoneval,Extruder\WObj:=Workobject_1;
MoveL RelTool (p1,80.500000,8.500000,9.000000,\Rx:=0.000000,\Ry:=0.000000),vel1,zoneval,Extruder\WObj:=Workobject_1;
MoveL RelTool (p1,78.000000,8.500000,9.000000,\Rx:=0.000000,\Ry:=0.000000),vel1,zoneval,Extruder\WObj:=Workobject_1;
MoveL RelTool (p1,75.500000,8.500000,9.000000,\Rx:=0.000000,\Ry:=0.000000),vel1,zoneval,Extruder\WObj:=Workobject_1;
MoveL RelTool (p1,73.000000,8.500000,9.000000,\Rx:=0.000000,\Ry:=0.000000),vel1,zoneval,Extruder\WObj:=Workobject_1;
MoveL RelTool (p1,70.500000,8.500000,9.000000,\Rx:=0.000000,\Ry:=0.000000),vel1,zoneval,Extruder\WObj:=Workobject_1;
MoveL RelTool (p1,68.000000,8.500000,9.192958,\Rx:=0.000000,\Ry:=6.326197),vel1,zoneval,Extruder\WObj:=Workobject_1;
MoveL RelTool (p1,65.500000,8.500000,11.706154,\Rx:=0.000000,\Ry:=9.902860),vel1,zoneval,Extruder\WObj:=Workobject_1;
MoveL RelTool (p1,63.000000,8.500000,13.771773,\Rx:=0.000000,\Ry:=7.227695),vel1,zoneval,Extruder\WObj:=Workobject_1;
MoveL RelTool (p1,60.500000,8.500000,15.226913,\Rx:=0.000000,\Ry:=6.061214),vel1,zoneval,Extruder\WObj:=Workobject_1;
MoveL RelTool (p1,58.000000,8.500000,16.345998,\Rx:=0.000000,\Ry:=5.005887),vel1,zoneval,Extruder\WObj:=Workobject_1;
MoveL RelTool (p1,55.500000,8.500000,17.210825,\Rx:=0.000000,\Ry:=4.006255),vel1,zoneval,Extruder\WObj:=Workobject_1;
MoveL RelTool (p1,53.000000,8.500000,17.871774,\Rx:=0.000000,\Ry:=3.108480),vel1,zoneval,Extruder\WObj:=Workobject_1;
MoveL RelTool (p1,50.500000,8.500000,18.361483,\Rx:=0.000000,\Ry:=2.217990),vel1,zoneval,Extruder\WObj:=Workobject_1;
MoveL RelTool (p1,48.000000,8.500000,18.701647,\Rx:=0.000000,\Ry:=1.375675),vel1,zoneval,Extruder\WObj:=Workobject_1;
MoveL RelTool (p1,45.500000,8.500000,18.907436,\Rx:=0.000000,\Ry:=0.547333),vel1,zoneval,Extruder\WObj:=Workobject_1;
MoveL RelTool (p1,43.000000,8.500000,18.993242,\Rx:=0.000000,\Ry:=-0.131676),vel1,zoneval,Extruder\WObj:=Workobject_1;
MoveL RelTool (p1,40.500000,8.500000,18.917003,\Rx:=0.000000,\Ry:=-0.809967),vel1,zoneval,Extruder\WObj:=Workobject_1;
MoveL RelTool (p1,38.000000,8.500000,18.733099,\Rx:=0.000000,\Ry:=-1.652509),vel1,zoneval,Extruder\WObj:=Workobject_1;
MoveL RelTool (p1,35.500000,8.500000,18.406795,\Rx:=0.000000,\Ry:=-2.278631),vel1,zoneval,Extruder\WObj:=Workobject_1;
MoveL RelTool (p1,33.000000,8.500000,17.912470,\Rx:=0.000000,\Ry:=-2.537038),vel1,zoneval,Extruder\WObj:=Workobject_1;
MoveL RelTool (p1,30.500000,8.500000,17.255542,\Rx:=0.000000,\Ry:=-3.471339),vel1,zoneval,Extruder\WObj:=Workobject_1;
MoveL RelTool (p1,28.000000,8.500000,16.406426,\Rx:=0.000000,\Ry:=-4.442626),vel1,zoneval,Extruder\WObj:=Workobject_1;
MoveL RelTool (p1,25.500000,8.500000,15.318735,\Rx:=0.000000,\Ry:=-5.751524),vel1,zoneval,Extruder\WObj:=Workobject_1;
MoveL RelTool (p1,23.000000,8.500000,13.890588,\Rx:=0.000000,\Ry:=-7.985654),vel1,zoneval,Extruder\WObj:=Workobject_1;
MoveL RelTool (p1,20.500000,8.500000,11.879398,\Rx:=0.000000,\Ry:=-10.154539),vel1,zoneval,Extruder\WObj:=Workobject_1;
MoveL RelTool (p1,18.000000,8.500000,9.264501,\Rx:=0.000000,\Ry:=-4.411855),vel1,zoneval,Extruder\WObj:=Workobject_1;
MoveL RelTool (p1,15.500000,8.500000,9.000000,\Rx:=0.000000,\Ry:=0.000000),vel1,zoneval,Extruder\WObj:=Workobject_1;
MoveL RelTool (p1,13.000000,8.500000,9.000000,\Rx:=0.000000,\Ry:=0.000000),vel1,zoneval,Extruder\WObj:=Workobject_1;
MoveL RelTool (p1,10.500000,8.500000,9.000000,\Rx:=0.000000,\Ry:=0.000000),vel1,zoneval,Extruder\WObj:=Workobject_1;
MoveL RelTool (p1,8.000000,8.500000,9.000000,\Rx:=0.000000,\Ry:=0.000000),vel1,zoneval,Extruder\WObj:=Workobject_1;
MoveL RelTool (p1,5.500000,8.500000,9.000000,\Rx:=0.000000,\Ry:=0.000000),vel1,zoneval,Extruder\WObj:=Workobject_1;
MoveL RelTool (p1,3.000000,8.500000,9.000000,\Rx:=0.000000,\Ry:=0.000000),vel1,zoneval,Extruder\WObj:=Workobject_1;
MoveL RelTool (p1,5.000000,9.000000,9.000000,\Rx:=0.000000,\Ry:=-0.000000),vel1,zoneval,Extruder\WObj:=Workobject_1;
MoveL RelTool (p1,7.500000,9.000000,9.000000,\Rx:=0.000000,\Ry:=-0.000000),vel1,zoneval,Extruder\WObj:=Workobject_1;
MoveL RelTool (p1,10.000000,9.000000,9.000000,\Rx:=0.000000,\Ry:=-0.000000),vel1,zoneval,Extruder\WObj:=Workobject_1;
MoveL RelTool (p1,12.500000,9.000000,9.000000,\Rx:=0.000000,\Ry:=-0.000000),vel1,zoneval,Extruder\WObj:=Workobject_1;
MoveL RelTool (p1,15.000000,9.000000,9.000000,\Rx:=0.000000,\Ry:=-0.000000),vel1,zoneval,Extruder\WObj:=Workobject_1;
MoveL RelTool (p1,17.500000,9.000000,9.083964,\Rx:=0.000000,\Ry:=-4.411855),vel1,zoneval,Extruder\WObj:=Workobject_1;
MoveL RelTool (p1,20.000000,9.000000,11.367111,\Rx:=0.000000,\Ry:=-10.154539),vel1,zoneval,Extruder\WObj:=Workobject_1;
MoveL RelTool (p1,22.500000,9.000000,13.528177,\Rx:=0.000000,\Ry:=-7.985654),vel1,zoneval,Extruder\WObj:=Workobject_1;
MoveL RelTool (p1,25.000000,9.000000,15.076143,\Rx:=0.000000,\Ry:=-5.751524),vel1,zoneval,Extruder\WObj:=Workobject_1;
MoveL RelTool (p1,27.500000,9.000000,16.224522,\Rx:=0.000000,\Ry:=-4.442626),vel1,zoneval,Extruder\WObj:=Workobject_1;
MoveL RelTool (p1,30.000000,9.000000,17.115741,\Rx:=0.000000,\Ry:=-3.471339),vel1,zoneval,Extruder\WObj:=Workobject_1;
MoveL RelTool (p1,32.500000,9.000000,17.811501,\Rx:=0.000000,\Ry:=-2.537038),vel1,zoneval,Extruder\WObj:=Workobject_1;
MoveL RelTool (p1,35.000000,9.000000,18.316346,\Rx:=0.000000,\Ry:=-2.278631),vel1,zoneval,Extruder\WObj:=Workobject_1;
MoveL RelTool (p1,37.500000,9.000000,18.667838,\Rx:=0.000000,\Ry:=-1.652509),vel1,zoneval,Extruder\WObj:=Workobject_1;
MoveL RelTool (p1,40.000000,9.000000,18.885153,\Rx:=0.000000,\Ry:=-0.809967),vel1,zoneval,Extruder\WObj:=Workobject_1;
MoveL RelTool (p1,42.500000,9.000000,18.988071,\Rx:=0.000000,\Ry:=-0.131676),vel1,zoneval,Extruder\WObj:=Workobject_1;
MoveL RelTool (p1,45.000000,9.000000,18.928943,\Rx:=0.000000,\Ry:=0.547333),vel1,zoneval,Extruder\WObj:=Workobject_1;
MoveL RelTool (p1,47.500000,9.000000,18.755880,\Rx:=0.000000,\Ry:=1.375675),vel1,zoneval,Extruder\WObj:=Workobject_1;
MoveL RelTool (p1,50.000000,9.000000,18.449475,\Rx:=0.000000,\Ry:=2.217990),vel1,zoneval,Extruder\WObj:=Workobject_1;
MoveL RelTool (p1,52.500000,9.000000,17.996328,\Rx:=0.000000,\Ry:=3.108480),vel1,zoneval,Extruder\WObj:=Workobject_1;
MoveL RelTool (p1,55.000000,9.000000,17.373557,\Rx:=0.000000,\Ry:=4.006255),vel1,zoneval,Extruder\WObj:=Workobject_1;
MoveL RelTool (p1,57.500000,9.000000,16.553376,\Rx:=0.000000,\Ry:=5.005887),vel1,zoneval,Extruder\WObj:=Workobject_1;
MoveL RelTool (p1,60.000000,9.000000,15.484711,\Rx:=0.000000,\Ry:=6.061214),vel1,zoneval,Extruder\WObj:=Workobject_1;
MoveL RelTool (p1,62.500000,9.000000,14.090610,\Rx:=0.000000,\Ry:=7.227695),vel1,zoneval,Extruder\WObj:=Workobject_1;
MoveL RelTool (p1,65.000000,9.000000,12.198583,\Rx:=0.000000,\Ry:=9.902860),vel1,zoneval,Extruder\WObj:=Workobject_1;
MoveL RelTool (p1,67.500000,9.000000,9.464073,\Rx:=0.000000,\Ry:=6.326197),vel1,zoneval,Extruder\WObj:=Workobject_1;
MoveL RelTool (p1,70.000000,9.000000,9.000000,\Rx:=0.000000,\Ry:=-0.000000),vel1,zoneval,Extruder\WObj:=Workobject_1;
MoveL RelTool (p1,72.500000,9.000000,9.000000,\Rx:=0.000000,\Ry:=-0.000000),vel1,zoneval,Extruder\WObj:=Workobject_1;
MoveL RelTool (p1,75.000000,9.000000,9.000000,\Rx:=0.000000,\Ry:=-0.000000),vel1,zoneval,Extruder\WObj:=Workobject_1;
MoveL RelTool (p1,77.500000,9.000000,9.000000,\Rx:=0.000000,\Ry:=-0.000000),vel1,zoneval,Extruder\WObj:=Workobject_1;
MoveL RelTool (p1,80.000000,9.000000,9.000000,\Rx:=0.000000,\Ry:=-0.000000),vel1,zoneval,Extruder\WObj:=Workobject_1;
MoveL RelTool (p1,82.500000,9.000000,9.000000,\Rx:=0.000000,\Ry:=-0.000000),vel1,zoneval,Extruder\WObj:=Workobject_1;
MoveL RelTool (p1,80.500000,9.500000,9.000000,\Rx:=0.000000,\Ry:=0.000000),vel1,zoneval,Extruder\WObj:=Workobject_1;
MoveL RelTool (p1,78.000000,9.500000,9.000000,\Rx:=0.000000,\Ry:=0.000000),vel1,zoneval,Extruder\WObj:=Workobject_1;
MoveL RelTool (p1,75.500000,9.500000,9.000000,\Rx:=0.000000,\Ry:=0.000000),vel1,zoneval,Extruder\WObj:=Workobject_1;
MoveL RelTool (p1,73.000000,9.500000,9.000000,\Rx:=0.000000,\Ry:=0.000000),vel1,zoneval,Extruder\WObj:=Workobject_1;
MoveL RelTool (p1,70.500000,9.500000,9.000000,\Rx:=0.000000,\Ry:=0.000000),vel1,zoneval,Extruder\WObj:=Workobject_1;
MoveL RelTool (p1,68.000000,9.500000,9.192958,\Rx:=0.000000,\Ry:=6.326197),vel1,zoneval,Extruder\WObj:=Workobject_1;
MoveL RelTool (p1,65.500000,9.500000,11.706154,\Rx:=0.000000,\Ry:=9.902860),vel1,zoneval,Extruder\WObj:=Workobject_1;
MoveL RelTool (p1,63.000000,9.500000,13.771773,\Rx:=0.000000,\Ry:=7.227695),vel1,zoneval,Extruder\WObj:=Workobject_1;
MoveL RelTool (p1,60.500000,9.500000,15.226913,\Rx:=0.000000,\Ry:=6.061214),vel1,zoneval,Extruder\WObj:=Workobject_1;
MoveL RelTool (p1,58.000000,9.500000,16.345998,\Rx:=0.000000,\Ry:=5.005887),vel1,zoneval,Extruder\WObj:=Workobject_1;
MoveL RelTool (p1,55.500000,9.500000,17.210825,\Rx:=0.000000,\Ry:=4.006255),vel1,zoneval,Extruder\WObj:=Workobject_1;
MoveL RelTool (p1,53.000000,9.500000,17.871774,\Rx:=0.000000,\Ry:=3.108480),vel1,zoneval,Extruder\WObj:=Workobject_1;
MoveL RelTool (p1,50.500000,9.500000,18.361483,\Rx:=0.000000,\Ry:=2.217990),vel1,zoneval,Extruder\WObj:=Workobject_1;
MoveL RelTool (p1,48.000000,9.500000,18.701647,\Rx:=0.000000,\Ry:=1.375675),vel1,zoneval,Extruder\WObj:=Workobject_1;
MoveL RelTool (p1,45.500000,9.500000,18.907436,\Rx:=0.000000,\Ry:=0.547333),vel1,zoneval,Extruder\WObj:=Workobject_1;
MoveL RelTool (p1,43.000000,9.500000,18.993242,\Rx:=0.000000,\Ry:=-0.131676),vel1,zoneval,Extruder\WObj:=Workobject_1;
MoveL RelTool (p1,40.500000,9.500000,18.917003,\Rx:=0.000000,\Ry:=-0.809967),vel1,zoneval,Extruder\WObj:=Workobject_1;
MoveL RelTool (p1,38.000000,9.500000,18.733099,\Rx:=0.000000,\Ry:=-1.652509),vel1,zoneval,Extruder\WObj:=Workobject_1;
MoveL RelTool (p1,35.500000,9.500000,18.406795,\Rx:=0.000000,\Ry:=-2.278631),vel1,zoneval,Extruder\WObj:=Workobject_1;
MoveL RelTool (p1,33.000000,9.500000,17.912470,\Rx:=0.000000,\Ry:=-2.537038),vel1,zoneval,Extruder\WObj:=Workobject_1;
MoveL RelTool (p1,30.500000,9.500000,17.255542,\Rx:=0.000000,\Ry:=-3.471339),vel1,zoneval,Extruder\WObj:=Workobject_1;
MoveL RelTool (p1,28.000000,9.500000,16.406426,\Rx:=0.000000,\Ry:=-4.442626),vel1,zoneval,Extruder\WObj:=Workobject_1;
MoveL RelTool (p1,25.500000,9.500000,15.318735,\Rx:=0.000000,\Ry:=-5.751524),vel1,zoneval,Extruder\WObj:=Workobject_1;
MoveL RelTool (p1,23.000000,9.500000,13.890588,\Rx:=0.000000,\Ry:=-7.985654),vel1,zoneval,Extruder\WObj:=Workobject_1;
MoveL RelTool (p1,20.500000,9.500000,11.879398,\Rx:=0.000000,\Ry:=-10.154539),vel1,zoneval,Extruder\WObj:=Workobject_1;
MoveL RelTool (p1,18.000000,9.500000,9.264501,\Rx:=0.000000,\Ry:=-4.411855),vel1,zoneval,Extruder\WObj:=Workobject_1;
MoveL RelTool (p1,15.500000,9.500000,9.000000,\Rx:=0.000000,\Ry:=0.000000),vel1,zoneval,Extruder\WObj:=Workobject_1;
MoveL RelTool (p1,13.000000,9.500000,9.000000,\Rx:=0.000000,\Ry:=0.000000),vel1,zoneval,Extruder\WObj:=Workobject_1;
MoveL RelTool (p1,10.500000,9.500000,9.000000,\Rx:=0.000000,\Ry:=0.000000),vel1,zoneval,Extruder\WObj:=Workobject_1;
MoveL RelTool (p1,8.000000,9.500000,9.000000,\Rx:=0.000000,\Ry:=0.000000),vel1,zoneval,Extruder\WObj:=Workobject_1;
MoveL RelTool (p1,5.500000,9.500000,9.000000,\Rx:=0.000000,\Ry:=0.000000),vel1,zoneval,Extruder\WObj:=Workobject_1;
MoveL RelTool (p1,3.000000,9.500000,9.000000,\Rx:=0.000000,\Ry:=0.000000),vel1,zoneval,Extruder\WObj:=Workobject_1;
MoveL RelTool (p1,5.000000,10.000000,9.000000,\Rx:=0.000000,\Ry:=-0.000000),vel1,zoneval,Extruder\WObj:=Workobject_1;
MoveL RelTool (p1,7.500000,10.000000,9.000000,\Rx:=0.000000,\Ry:=-0.000000),vel1,zoneval,Extruder\WObj:=Workobject_1;
MoveL RelTool (p1,10.000000,10.000000,9.000000,\Rx:=0.000000,\Ry:=-0.000000),vel1,zoneval,Extruder\WObj:=Workobject_1;
MoveL RelTool (p1,12.500000,10.000000,9.000000,\Rx:=0.000000,\Ry:=-0.000000),vel1,zoneval,Extruder\WObj:=Workobject_1;
MoveL RelTool (p1,15.000000,10.000000,9.000000,\Rx:=0.000000,\Ry:=-0.000000),vel1,zoneval,Extruder\WObj:=Workobject_1;
MoveL RelTool (p1,17.500000,10.000000,9.083964,\Rx:=0.000000,\Ry:=-4.411855),vel1,zoneval,Extruder\WObj:=Workobject_1;
MoveL RelTool (p1,20.000000,10.000000,11.367111,\Rx:=0.000000,\Ry:=-10.154539),vel1,zoneval,Extruder\WObj:=Workobject_1;
MoveL RelTool (p1,22.500000,10.000000,13.528177,\Rx:=0.000000,\Ry:=-7.985654),vel1,zoneval,Extruder\WObj:=Workobject_1;
MoveL RelTool (p1,25.000000,10.000000,15.076143,\Rx:=0.000000,\Ry:=-5.751524),vel1,zoneval,Extruder\WObj:=Workobject_1;
MoveL RelTool (p1,27.500000,10.000000,16.224522,\Rx:=0.000000,\Ry:=-4.442626),vel1,zoneval,Extruder\WObj:=Workobject_1;
MoveL RelTool (p1,30.000000,10.000000,17.115741,\Rx:=0.000000,\Ry:=-3.471339),vel1,zoneval,Extruder\WObj:=Workobject_1;
MoveL RelTool (p1,32.500000,10.000000,17.811501,\Rx:=0.000000,\Ry:=-2.537038),vel1,zoneval,Extruder\WObj:=Workobject_1;
MoveL RelTool (p1,35.000000,10.000000,18.316346,\Rx:=0.000000,\Ry:=-2.278631),vel1,zoneval,Extruder\WObj:=Workobject_1;
MoveL RelTool (p1,37.500000,10.000000,18.667838,\Rx:=0.000000,\Ry:=-1.652509),vel1,zoneval,Extruder\WObj:=Workobject_1;
MoveL RelTool (p1,40.000000,10.000000,18.885153,\Rx:=0.000000,\Ry:=-0.809967),vel1,zoneval,Extruder\WObj:=Workobject_1;
MoveL RelTool (p1,42.500000,10.000000,18.988071,\Rx:=0.000000,\Ry:=-0.131676),vel1,zoneval,Extruder\WObj:=Workobject_1;
MoveL RelTool (p1,45.000000,10.000000,18.928943,\Rx:=0.000000,\Ry:=0.547333),vel1,zoneval,Extruder\WObj:=Workobject_1;
MoveL RelTool (p1,47.500000,10.000000,18.755880,\Rx:=0.000000,\Ry:=1.375675),vel1,zoneval,Extruder\WObj:=Workobject_1;
MoveL RelTool (p1,50.000000,10.000000,18.449475,\Rx:=0.000000,\Ry:=2.217990),vel1,zoneval,Extruder\WObj:=Workobject_1;
MoveL RelTool (p1,52.500000,10.000000,17.996328,\Rx:=0.000000,\Ry:=3.108480),vel1,zoneval,Extruder\WObj:=Workobject_1;
MoveL RelTool (p1,55.000000,10.000000,17.373557,\Rx:=0.000000,\Ry:=4.006255),vel1,zoneval,Extruder\WObj:=Workobject_1;
MoveL RelTool (p1,57.500000,10.000000,16.553376,\Rx:=0.000000,\Ry:=5.005887),vel1,zoneval,Extruder\WObj:=Workobject_1;
MoveL RelTool (p1,60.000000,10.000000,15.484711,\Rx:=0.000000,\Ry:=6.061214),vel1,zoneval,Extruder\WObj:=Workobject_1;
MoveL RelTool (p1,62.500000,10.000000,14.090610,\Rx:=0.000000,\Ry:=7.227695),vel1,zoneval,Extruder\WObj:=Workobject_1;
MoveL RelTool (p1,65.000000,10.000000,12.198583,\Rx:=0.000000,\Ry:=9.902860),vel1,zoneval,Extruder\WObj:=Workobject_1;
MoveL RelTool (p1,67.500000,10.000000,9.464073,\Rx:=0.000000,\Ry:=6.326197),vel1,zoneval,Extruder\WObj:=Workobject_1;
MoveL RelTool (p1,70.000000,10.000000,9.000000,\Rx:=0.000000,\Ry:=-0.000000),vel1,zoneval,Extruder\WObj:=Workobject_1;
MoveL RelTool (p1,72.500000,10.000000,9.000000,\Rx:=0.000000,\Ry:=-0.000000),vel1,zoneval,Extruder\WObj:=Workobject_1;
MoveL RelTool (p1,75.000000,10.000000,9.000000,\Rx:=0.000000,\Ry:=-0.000000),vel1,zoneval,Extruder\WObj:=Workobject_1;
MoveL RelTool (p1,77.500000,10.000000,9.000000,\Rx:=0.000000,\Ry:=-0.000000),vel1,zoneval,Extruder\WObj:=Workobject_1;
MoveL RelTool (p1,80.000000,10.000000,9.000000,\Rx:=0.000000,\Ry:=-0.000000),vel1,zoneval,Extruder\WObj:=Workobject_1;
MoveL RelTool (p1,82.500000,10.000000,9.000000,\Rx:=0.000000,\Ry:=-0.000000),vel1,zoneval,Extruder\WObj:=Workobject_1;
MoveL RelTool (p1,80.500000,10.500000,9.000000,\Rx:=0.000000,\Ry:=0.000000),vel1,zoneval,Extruder\WObj:=Workobject_1;
MoveL RelTool (p1,78.000000,10.500000,9.000000,\Rx:=0.000000,\Ry:=0.000000),vel1,zoneval,Extruder\WObj:=Workobject_1;
MoveL RelTool (p1,75.500000,10.500000,9.000000,\Rx:=0.000000,\Ry:=0.000000),vel1,zoneval,Extruder\WObj:=Workobject_1;
MoveL RelTool (p1,73.000000,10.500000,9.000000,\Rx:=0.000000,\Ry:=0.000000),vel1,zoneval,Extruder\WObj:=Workobject_1;
MoveL RelTool (p1,70.500000,10.500000,9.000000,\Rx:=0.000000,\Ry:=0.000000),vel1,zoneval,Extruder\WObj:=Workobject_1;
MoveL RelTool (p1,68.000000,10.500000,9.192958,\Rx:=0.000000,\Ry:=6.326197),vel1,zoneval,Extruder\WObj:=Workobject_1;
MoveL RelTool (p1,65.500000,10.500000,11.706154,\Rx:=0.000000,\Ry:=9.902860),vel1,zoneval,Extruder\WObj:=Workobject_1;
MoveL RelTool (p1,63.000000,10.500000,13.771773,\Rx:=0.000000,\Ry:=7.227695),vel1,zoneval,Extruder\WObj:=Workobject_1;
MoveL RelTool (p1,60.500000,10.500000,15.226913,\Rx:=0.000000,\Ry:=6.061214),vel1,zoneval,Extruder\WObj:=Workobject_1;
MoveL RelTool (p1,58.000000,10.500000,16.345998,\Rx:=0.000000,\Ry:=5.005887),vel1,zoneval,Extruder\WObj:=Workobject_1;
MoveL RelTool (p1,55.500000,10.500000,17.210825,\Rx:=0.000000,\Ry:=4.006255),vel1,zoneval,Extruder\WObj:=Workobject_1;
MoveL RelTool (p1,53.000000,10.500000,17.871774,\Rx:=0.000000,\Ry:=3.108480),vel1,zoneval,Extruder\WObj:=Workobject_1;
MoveL RelTool (p1,50.500000,10.500000,18.361483,\Rx:=0.000000,\Ry:=2.217990),vel1,zoneval,Extruder\WObj:=Workobject_1;
MoveL RelTool (p1,48.000000,10.500000,18.701647,\Rx:=0.000000,\Ry:=1.375675),vel1,zoneval,Extruder\WObj:=Workobject_1;
MoveL RelTool (p1,45.500000,10.500000,18.907436,\Rx:=0.000000,\Ry:=0.547333),vel1,zoneval,Extruder\WObj:=Workobject_1;
MoveL RelTool (p1,43.000000,10.500000,18.993242,\Rx:=0.000000,\Ry:=-0.131676),vel1,zoneval,Extruder\WObj:=Workobject_1;
MoveL RelTool (p1,40.500000,10.500000,18.917003,\Rx:=0.000000,\Ry:=-0.809967),vel1,zoneval,Extruder\WObj:=Workobject_1;
MoveL RelTool (p1,38.000000,10.500000,18.733099,\Rx:=0.000000,\Ry:=-1.652509),vel1,zoneval,Extruder\WObj:=Workobject_1;
MoveL RelTool (p1,35.500000,10.500000,18.406795,\Rx:=0.000000,\Ry:=-2.278631),vel1,zoneval,Extruder\WObj:=Workobject_1;
MoveL RelTool (p1,33.000000,10.500000,17.912470,\Rx:=0.000000,\Ry:=-2.537038),vel1,zoneval,Extruder\WObj:=Workobject_1;
MoveL RelTool (p1,30.500000,10.500000,17.255542,\Rx:=0.000000,\Ry:=-3.471339),vel1,zoneval,Extruder\WObj:=Workobject_1;
MoveL RelTool (p1,28.000000,10.500000,16.406426,\Rx:=0.000000,\Ry:=-4.442626),vel1,zoneval,Extruder\WObj:=Workobject_1;
MoveL RelTool (p1,25.500000,10.500000,15.318735,\Rx:=0.000000,\Ry:=-5.751524),vel1,zoneval,Extruder\WObj:=Workobject_1;
MoveL RelTool (p1,23.000000,10.500000,13.890588,\Rx:=0.000000,\Ry:=-7.985654),vel1,zoneval,Extruder\WObj:=Workobject_1;
MoveL RelTool (p1,20.500000,10.500000,11.879398,\Rx:=0.000000,\Ry:=-10.154539),vel1,zoneval,Extruder\WObj:=Workobject_1;
MoveL RelTool (p1,18.000000,10.500000,9.264501,\Rx:=0.000000,\Ry:=-4.411855),vel1,zoneval,Extruder\WObj:=Workobject_1;
MoveL RelTool (p1,15.500000,10.500000,9.000000,\Rx:=0.000000,\Ry:=0.000000),vel1,zoneval,Extruder\WObj:=Workobject_1;
MoveL RelTool (p1,13.000000,10.500000,9.000000,\Rx:=0.000000,\Ry:=0.000000),vel1,zoneval,Extruder\WObj:=Workobject_1;
MoveL RelTool (p1,10.500000,10.500000,9.000000,\Rx:=0.000000,\Ry:=0.000000),vel1,zoneval,Extruder\WObj:=Workobject_1;
MoveL RelTool (p1,8.000000,10.500000,9.000000,\Rx:=0.000000,\Ry:=0.000000),vel1,zoneval,Extruder\WObj:=Workobject_1;
MoveL RelTool (p1,5.500000,10.500000,9.000000,\Rx:=0.000000,\Ry:=0.000000),vel1,zoneval,Extruder\WObj:=Workobject_1;
MoveL RelTool (p1,3.000000,10.500000,9.000000,\Rx:=0.000000,\Ry:=0.000000),vel1,zoneval,Extruder\WObj:=Workobject_1;
MoveL RelTool (p1,5.000000,11.000000,9.000000,\Rx:=0.000000,\Ry:=-0.000000),vel1,zoneval,Extruder\WObj:=Workobject_1;
MoveL RelTool (p1,7.500000,11.000000,9.000000,\Rx:=0.000000,\Ry:=-0.000000),vel1,zoneval,Extruder\WObj:=Workobject_1;
MoveL RelTool (p1,10.000000,11.000000,9.000000,\Rx:=0.000000,\Ry:=-0.000000),vel1,zoneval,Extruder\WObj:=Workobject_1;
MoveL RelTool (p1,12.500000,11.000000,9.000000,\Rx:=0.000000,\Ry:=-0.000000),vel1,zoneval,Extruder\WObj:=Workobject_1;
MoveL RelTool (p1,15.000000,11.000000,9.000000,\Rx:=0.000000,\Ry:=-0.000000),vel1,zoneval,Extruder\WObj:=Workobject_1;
MoveL RelTool (p1,17.500000,11.000000,9.083964,\Rx:=0.000000,\Ry:=-4.411855),vel1,zoneval,Extruder\WObj:=Workobject_1;
MoveL RelTool (p1,20.000000,11.000000,11.367111,\Rx:=0.000000,\Ry:=-10.154539),vel1,zoneval,Extruder\WObj:=Workobject_1;
MoveL RelTool (p1,22.500000,11.000000,13.528177,\Rx:=0.000000,\Ry:=-7.985654),vel1,zoneval,Extruder\WObj:=Workobject_1;
MoveL RelTool (p1,25.000000,11.000000,15.076143,\Rx:=0.000000,\Ry:=-5.751524),vel1,zoneval,Extruder\WObj:=Workobject_1;
MoveL RelTool (p1,27.500000,11.000000,16.224522,\Rx:=0.000000,\Ry:=-4.442626),vel1,zoneval,Extruder\WObj:=Workobject_1;
MoveL RelTool (p1,30.000000,11.000000,17.115741,\Rx:=0.000000,\Ry:=-3.471339),vel1,zoneval,Extruder\WObj:=Workobject_1;
MoveL RelTool (p1,32.500000,11.000000,17.811501,\Rx:=0.000000,\Ry:=-2.537038),vel1,zoneval,Extruder\WObj:=Workobject_1;
MoveL RelTool (p1,35.000000,11.000000,18.316346,\Rx:=0.000000,\Ry:=-2.278631),vel1,zoneval,Extruder\WObj:=Workobject_1;
MoveL RelTool (p1,37.500000,11.000000,18.667838,\Rx:=0.000000,\Ry:=-1.652509),vel1,zoneval,Extruder\WObj:=Workobject_1;
MoveL RelTool (p1,40.000000,11.000000,18.885153,\Rx:=0.000000,\Ry:=-0.809967),vel1,zoneval,Extruder\WObj:=Workobject_1;
MoveL RelTool (p1,42.500000,11.000000,18.988071,\Rx:=0.000000,\Ry:=-0.131676),vel1,zoneval,Extruder\WObj:=Workobject_1;
MoveL RelTool (p1,45.000000,11.000000,18.928943,\Rx:=0.000000,\Ry:=0.547333),vel1,zoneval,Extruder\WObj:=Workobject_1;
MoveL RelTool (p1,47.500000,11.000000,18.755880,\Rx:=0.000000,\Ry:=1.375675),vel1,zoneval,Extruder\WObj:=Workobject_1;
MoveL RelTool (p1,50.000000,11.000000,18.449475,\Rx:=0.000000,\Ry:=2.217990),vel1,zoneval,Extruder\WObj:=Workobject_1;
MoveL RelTool (p1,52.500000,11.000000,17.996328,\Rx:=0.000000,\Ry:=3.108480),vel1,zoneval,Extruder\WObj:=Workobject_1;
MoveL RelTool (p1,55.000000,11.000000,17.373557,\Rx:=0.000000,\Ry:=4.006255),vel1,zoneval,Extruder\WObj:=Workobject_1;
MoveL RelTool (p1,57.500000,11.000000,16.553376,\Rx:=0.000000,\Ry:=5.005887),vel1,zoneval,Extruder\WObj:=Workobject_1;
MoveL RelTool (p1,60.000000,11.000000,15.484711,\Rx:=0.000000,\Ry:=6.061214),vel1,zoneval,Extruder\WObj:=Workobject_1;
MoveL RelTool (p1,62.500000,11.000000,14.090610,\Rx:=0.000000,\Ry:=7.227695),vel1,zoneval,Extruder\WObj:=Workobject_1;
MoveL RelTool (p1,65.000000,11.000000,12.198583,\Rx:=0.000000,\Ry:=9.902860),vel1,zoneval,Extruder\WObj:=Workobject_1;
MoveL RelTool (p1,67.500000,11.000000,9.464073,\Rx:=0.000000,\Ry:=6.326197),vel1,zoneval,Extruder\WObj:=Workobject_1;
MoveL RelTool (p1,70.000000,11.000000,9.000000,\Rx:=0.000000,\Ry:=-0.000000),vel1,zoneval,Extruder\WObj:=Workobject_1;
MoveL RelTool (p1,72.500000,11.000000,9.000000,\Rx:=0.000000,\Ry:=-0.000000),vel1,zoneval,Extruder\WObj:=Workobject_1;
MoveL RelTool (p1,75.000000,11.000000,9.000000,\Rx:=0.000000,\Ry:=-0.000000),vel1,zoneval,Extruder\WObj:=Workobject_1;
MoveL RelTool (p1,77.500000,11.000000,9.000000,\Rx:=0.000000,\Ry:=-0.000000),vel1,zoneval,Extruder\WObj:=Workobject_1;
MoveL RelTool (p1,80.000000,11.000000,9.000000,\Rx:=0.000000,\Ry:=-0.000000),vel1,zoneval,Extruder\WObj:=Workobject_1;
MoveL RelTool (p1,82.500000,11.000000,9.000000,\Rx:=0.000000,\Ry:=-0.000000),vel1,zoneval,Extruder\WObj:=Workobject_1;
MoveL RelTool (p1,80.500000,11.500000,9.000000,\Rx:=0.000000,\Ry:=0.000000),vel1,zoneval,Extruder\WObj:=Workobject_1;
MoveL RelTool (p1,78.000000,11.500000,9.000000,\Rx:=0.000000,\Ry:=0.000000),vel1,zoneval,Extruder\WObj:=Workobject_1;
MoveL RelTool (p1,75.500000,11.500000,9.000000,\Rx:=0.000000,\Ry:=0.000000),vel1,zoneval,Extruder\WObj:=Workobject_1;
MoveL RelTool (p1,73.000000,11.500000,9.000000,\Rx:=0.000000,\Ry:=0.000000),vel1,zoneval,Extruder\WObj:=Workobject_1;
MoveL RelTool (p1,70.500000,11.500000,9.000000,\Rx:=0.000000,\Ry:=0.000000),vel1,zoneval,Extruder\WObj:=Workobject_1;
MoveL RelTool (p1,68.000000,11.500000,9.192958,\Rx:=0.000000,\Ry:=6.326197),vel1,zoneval,Extruder\WObj:=Workobject_1;
MoveL RelTool (p1,65.500000,11.500000,11.706154,\Rx:=0.000000,\Ry:=9.902860),vel1,zoneval,Extruder\WObj:=Workobject_1;
MoveL RelTool (p1,63.000000,11.500000,13.771773,\Rx:=0.000000,\Ry:=7.227695),vel1,zoneval,Extruder\WObj:=Workobject_1;
MoveL RelTool (p1,60.500000,11.500000,15.226913,\Rx:=0.000000,\Ry:=6.061214),vel1,zoneval,Extruder\WObj:=Workobject_1;
MoveL RelTool (p1,58.000000,11.500000,16.345998,\Rx:=0.000000,\Ry:=5.005887),vel1,zoneval,Extruder\WObj:=Workobject_1;
MoveL RelTool (p1,55.500000,11.500000,17.210825,\Rx:=0.000000,\Ry:=4.006255),vel1,zoneval,Extruder\WObj:=Workobject_1;
MoveL RelTool (p1,53.000000,11.500000,17.871774,\Rx:=0.000000,\Ry:=3.108480),vel1,zoneval,Extruder\WObj:=Workobject_1;
MoveL RelTool (p1,50.500000,11.500000,18.361483,\Rx:=0.000000,\Ry:=2.217990),vel1,zoneval,Extruder\WObj:=Workobject_1;
MoveL RelTool (p1,48.000000,11.500000,18.701647,\Rx:=0.000000,\Ry:=1.375675),vel1,zoneval,Extruder\WObj:=Workobject_1;
MoveL RelTool (p1,45.500000,11.500000,18.907436,\Rx:=0.000000,\Ry:=0.547333),vel1,zoneval,Extruder\WObj:=Workobject_1;
MoveL RelTool (p1,43.000000,11.500000,18.993242,\Rx:=0.000000,\Ry:=-0.131676),vel1,zoneval,Extruder\WObj:=Workobject_1;
MoveL RelTool (p1,40.500000,11.500000,18.917003,\Rx:=0.000000,\Ry:=-0.809967),vel1,zoneval,Extruder\WObj:=Workobject_1;
MoveL RelTool (p1,38.000000,11.500000,18.733099,\Rx:=0.000000,\Ry:=-1.652509),vel1,zoneval,Extruder\WObj:=Workobject_1;
MoveL RelTool (p1,35.500000,11.500000,18.406795,\Rx:=0.000000,\Ry:=-2.278631),vel1,zoneval,Extruder\WObj:=Workobject_1;
MoveL RelTool (p1,33.000000,11.500000,17.912470,\Rx:=0.000000,\Ry:=-2.537038),vel1,zoneval,Extruder\WObj:=Workobject_1;
MoveL RelTool (p1,30.500000,11.500000,17.255542,\Rx:=0.000000,\Ry:=-3.471339),vel1,zoneval,Extruder\WObj:=Workobject_1;
MoveL RelTool (p1,28.000000,11.500000,16.406426,\Rx:=0.000000,\Ry:=-4.442626),vel1,zoneval,Extruder\WObj:=Workobject_1;
MoveL RelTool (p1,25.500000,11.500000,15.318735,\Rx:=0.000000,\Ry:=-5.751524),vel1,zoneval,Extruder\WObj:=Workobject_1;
MoveL RelTool (p1,23.000000,11.500000,13.890588,\Rx:=0.000000,\Ry:=-7.985654),vel1,zoneval,Extruder\WObj:=Workobject_1;
MoveL RelTool (p1,20.500000,11.500000,11.879398,\Rx:=0.000000,\Ry:=-10.154539),vel1,zoneval,Extruder\WObj:=Workobject_1;
MoveL RelTool (p1,18.000000,11.500000,9.264501,\Rx:=0.000000,\Ry:=-4.411855),vel1,zoneval,Extruder\WObj:=Workobject_1;
MoveL RelTool (p1,15.500000,11.500000,9.000000,\Rx:=0.000000,\Ry:=0.000000),vel1,zoneval,Extruder\WObj:=Workobject_1;
MoveL RelTool (p1,13.000000,11.500000,9.000000,\Rx:=0.000000,\Ry:=0.000000),vel1,zoneval,Extruder\WObj:=Workobject_1;
MoveL RelTool (p1,10.500000,11.500000,9.000000,\Rx:=0.000000,\Ry:=0.000000),vel1,zoneval,Extruder\WObj:=Workobject_1;
MoveL RelTool (p1,8.000000,11.500000,9.000000,\Rx:=0.000000,\Ry:=0.000000),vel1,zoneval,Extruder\WObj:=Workobject_1;
MoveL RelTool (p1,5.500000,11.500000,9.000000,\Rx:=0.000000,\Ry:=0.000000),vel1,zoneval,Extruder\WObj:=Workobject_1;
MoveL RelTool (p1,3.000000,11.500000,9.000000,\Rx:=0.000000,\Ry:=0.000000),vel1,zoneval,Extruder\WObj:=Workobject_1;
MoveL RelTool (p1,5.000000,12.000000,9.000000,\Rx:=0.000000,\Ry:=-0.000000),vel1,zoneval,Extruder\WObj:=Workobject_1;
MoveL RelTool (p1,7.500000,12.000000,9.000000,\Rx:=0.000000,\Ry:=-0.000000),vel1,zoneval,Extruder\WObj:=Workobject_1;
MoveL RelTool (p1,10.000000,12.000000,9.000000,\Rx:=0.000000,\Ry:=-0.000000),vel1,zoneval,Extruder\WObj:=Workobject_1;
MoveL RelTool (p1,12.500000,12.000000,9.000000,\Rx:=0.000000,\Ry:=-0.000000),vel1,zoneval,Extruder\WObj:=Workobject_1;
MoveL RelTool (p1,15.000000,12.000000,9.000000,\Rx:=0.000000,\Ry:=-0.000000),vel1,zoneval,Extruder\WObj:=Workobject_1;
MoveL RelTool (p1,17.500000,12.000000,9.083964,\Rx:=0.000000,\Ry:=-4.411855),vel1,zoneval,Extruder\WObj:=Workobject_1;
MoveL RelTool (p1,20.000000,12.000000,11.367111,\Rx:=0.000000,\Ry:=-10.154539),vel1,zoneval,Extruder\WObj:=Workobject_1;
MoveL RelTool (p1,22.500000,12.000000,13.528177,\Rx:=0.000000,\Ry:=-7.985654),vel1,zoneval,Extruder\WObj:=Workobject_1;
MoveL RelTool (p1,25.000000,12.000000,15.076143,\Rx:=0.000000,\Ry:=-5.751524),vel1,zoneval,Extruder\WObj:=Workobject_1;
MoveL RelTool (p1,27.500000,12.000000,16.224522,\Rx:=0.000000,\Ry:=-4.442626),vel1,zoneval,Extruder\WObj:=Workobject_1;
MoveL RelTool (p1,30.000000,12.000000,17.115741,\Rx:=0.000000,\Ry:=-3.471339),vel1,zoneval,Extruder\WObj:=Workobject_1;
MoveL RelTool (p1,32.500000,12.000000,17.811501,\Rx:=0.000000,\Ry:=-2.537038),vel1,zoneval,Extruder\WObj:=Workobject_1;
MoveL RelTool (p1,35.000000,12.000000,18.316346,\Rx:=0.000000,\Ry:=-2.278631),vel1,zoneval,Extruder\WObj:=Workobject_1;
MoveL RelTool (p1,37.500000,12.000000,18.667838,\Rx:=0.000000,\Ry:=-1.652509),vel1,zoneval,Extruder\WObj:=Workobject_1;
MoveL RelTool (p1,40.000000,12.000000,18.885153,\Rx:=0.000000,\Ry:=-0.809967),vel1,zoneval,Extruder\WObj:=Workobject_1;
MoveL RelTool (p1,42.500000,12.000000,18.988071,\Rx:=0.000000,\Ry:=-0.131676),vel1,zoneval,Extruder\WObj:=Workobject_1;
MoveL RelTool (p1,45.000000,12.000000,18.928943,\Rx:=0.000000,\Ry:=0.547333),vel1,zoneval,Extruder\WObj:=Workobject_1;
MoveL RelTool (p1,47.500000,12.000000,18.755880,\Rx:=0.000000,\Ry:=1.375675),vel1,zoneval,Extruder\WObj:=Workobject_1;
MoveL RelTool (p1,50.000000,12.000000,18.449475,\Rx:=0.000000,\Ry:=2.217990),vel1,zoneval,Extruder\WObj:=Workobject_1;
MoveL RelTool (p1,52.500000,12.000000,17.996328,\Rx:=0.000000,\Ry:=3.108480),vel1,zoneval,Extruder\WObj:=Workobject_1;
MoveL RelTool (p1,55.000000,12.000000,17.373557,\Rx:=0.000000,\Ry:=4.006255),vel1,zoneval,Extruder\WObj:=Workobject_1;
MoveL RelTool (p1,57.500000,12.000000,16.553376,\Rx:=0.000000,\Ry:=5.005887),vel1,zoneval,Extruder\WObj:=Workobject_1;
MoveL RelTool (p1,60.000000,12.000000,15.484711,\Rx:=0.000000,\Ry:=6.061214),vel1,zoneval,Extruder\WObj:=Workobject_1;
MoveL RelTool (p1,62.500000,12.000000,14.090610,\Rx:=0.000000,\Ry:=7.227695),vel1,zoneval,Extruder\WObj:=Workobject_1;
MoveL RelTool (p1,65.000000,12.000000,12.198583,\Rx:=0.000000,\Ry:=9.902860),vel1,zoneval,Extruder\WObj:=Workobject_1;
MoveL RelTool (p1,67.500000,12.000000,9.464073,\Rx:=0.000000,\Ry:=6.326197),vel1,zoneval,Extruder\WObj:=Workobject_1;
MoveL RelTool (p1,70.000000,12.000000,9.000000,\Rx:=0.000000,\Ry:=-0.000000),vel1,zoneval,Extruder\WObj:=Workobject_1;
MoveL RelTool (p1,72.500000,12.000000,9.000000,\Rx:=0.000000,\Ry:=-0.000000),vel1,zoneval,Extruder\WObj:=Workobject_1;
MoveL RelTool (p1,75.000000,12.000000,9.000000,\Rx:=0.000000,\Ry:=-0.000000),vel1,zoneval,Extruder\WObj:=Workobject_1;
MoveL RelTool (p1,77.500000,12.000000,9.000000,\Rx:=0.000000,\Ry:=-0.000000),vel1,zoneval,Extruder\WObj:=Workobject_1;
MoveL RelTool (p1,80.000000,12.000000,9.000000,\Rx:=0.000000,\Ry:=-0.000000),vel1,zoneval,Extruder\WObj:=Workobject_1;
MoveL RelTool (p1,82.500000,12.000000,9.000000,\Rx:=0.000000,\Ry:=-0.000000),vel1,zoneval,Extruder\WObj:=Workobject_1;
MoveL RelTool (p1,80.500000,12.500000,9.000000,\Rx:=0.000000,\Ry:=0.000000),vel1,zoneval,Extruder\WObj:=Workobject_1;
MoveL RelTool (p1,78.000000,12.500000,9.000000,\Rx:=0.000000,\Ry:=0.000000),vel1,zoneval,Extruder\WObj:=Workobject_1;
MoveL RelTool (p1,75.500000,12.500000,9.000000,\Rx:=0.000000,\Ry:=0.000000),vel1,zoneval,Extruder\WObj:=Workobject_1;
MoveL RelTool (p1,73.000000,12.500000,9.000000,\Rx:=0.000000,\Ry:=0.000000),vel1,zoneval,Extruder\WObj:=Workobject_1;
MoveL RelTool (p1,70.500000,12.500000,9.000000,\Rx:=0.000000,\Ry:=0.000000),vel1,zoneval,Extruder\WObj:=Workobject_1;
MoveL RelTool (p1,68.000000,12.500000,9.192958,\Rx:=0.000000,\Ry:=6.326197),vel1,zoneval,Extruder\WObj:=Workobject_1;
MoveL RelTool (p1,65.500000,12.500000,11.706154,\Rx:=0.000000,\Ry:=9.902860),vel1,zoneval,Extruder\WObj:=Workobject_1;
MoveL RelTool (p1,63.000000,12.500000,13.771773,\Rx:=0.000000,\Ry:=7.227695),vel1,zoneval,Extruder\WObj:=Workobject_1;
MoveL RelTool (p1,60.500000,12.500000,15.226913,\Rx:=0.000000,\Ry:=6.061214),vel1,zoneval,Extruder\WObj:=Workobject_1;
MoveL RelTool (p1,58.000000,12.500000,16.345998,\Rx:=0.000000,\Ry:=5.005887),vel1,zoneval,Extruder\WObj:=Workobject_1;
MoveL RelTool (p1,55.500000,12.500000,17.210825,\Rx:=0.000000,\Ry:=4.006255),vel1,zoneval,Extruder\WObj:=Workobject_1;
MoveL RelTool (p1,53.000000,12.500000,17.871774,\Rx:=0.000000,\Ry:=3.108480),vel1,zoneval,Extruder\WObj:=Workobject_1;
MoveL RelTool (p1,50.500000,12.500000,18.361483,\Rx:=0.000000,\Ry:=2.217990),vel1,zoneval,Extruder\WObj:=Workobject_1;
MoveL RelTool (p1,48.000000,12.500000,18.701647,\Rx:=0.000000,\Ry:=1.375675),vel1,zoneval,Extruder\WObj:=Workobject_1;
MoveL RelTool (p1,45.500000,12.500000,18.907436,\Rx:=0.000000,\Ry:=0.547333),vel1,zoneval,Extruder\WObj:=Workobject_1;
MoveL RelTool (p1,43.000000,12.500000,18.993242,\Rx:=0.000000,\Ry:=-0.131676),vel1,zoneval,Extruder\WObj:=Workobject_1;
MoveL RelTool (p1,40.500000,12.500000,18.917003,\Rx:=0.000000,\Ry:=-0.809967),vel1,zoneval,Extruder\WObj:=Workobject_1;
MoveL RelTool (p1,38.000000,12.500000,18.733099,\Rx:=0.000000,\Ry:=-1.652509),vel1,zoneval,Extruder\WObj:=Workobject_1;
MoveL RelTool (p1,35.500000,12.500000,18.406795,\Rx:=0.000000,\Ry:=-2.278631),vel1,zoneval,Extruder\WObj:=Workobject_1;
MoveL RelTool (p1,33.000000,12.500000,17.912470,\Rx:=0.000000,\Ry:=-2.537038),vel1,zoneval,Extruder\WObj:=Workobject_1;
MoveL RelTool (p1,30.500000,12.500000,17.255542,\Rx:=0.000000,\Ry:=-3.471339),vel1,zoneval,Extruder\WObj:=Workobject_1;
MoveL RelTool (p1,28.000000,12.500000,16.406426,\Rx:=0.000000,\Ry:=-4.442626),vel1,zoneval,Extruder\WObj:=Workobject_1;
MoveL RelTool (p1,25.500000,12.500000,15.318735,\Rx:=0.000000,\Ry:=-5.751524),vel1,zoneval,Extruder\WObj:=Workobject_1;
MoveL RelTool (p1,23.000000,12.500000,13.890588,\Rx:=0.000000,\Ry:=-7.985654),vel1,zoneval,Extruder\WObj:=Workobject_1;
MoveL RelTool (p1,20.500000,12.500000,11.879398,\Rx:=0.000000,\Ry:=-10.154539),vel1,zoneval,Extruder\WObj:=Workobject_1;
MoveL RelTool (p1,18.000000,12.500000,9.264501,\Rx:=0.000000,\Ry:=-4.411855),vel1,zoneval,Extruder\WObj:=Workobject_1;
MoveL RelTool (p1,15.500000,12.500000,9.000000,\Rx:=0.000000,\Ry:=0.000000),vel1,zoneval,Extruder\WObj:=Workobject_1;
MoveL RelTool (p1,13.000000,12.500000,9.000000,\Rx:=0.000000,\Ry:=0.000000),vel1,zoneval,Extruder\WObj:=Workobject_1;
MoveL RelTool (p1,10.500000,12.500000,9.000000,\Rx:=0.000000,\Ry:=0.000000),vel1,zoneval,Extruder\WObj:=Workobject_1;
MoveL RelTool (p1,8.000000,12.500000,9.000000,\Rx:=0.000000,\Ry:=0.000000),vel1,zoneval,Extruder\WObj:=Workobject_1;
MoveL RelTool (p1,5.500000,12.500000,9.000000,\Rx:=0.000000,\Ry:=0.000000),vel1,zoneval,Extruder\WObj:=Workobject_1;
MoveL RelTool (p1,3.000000,12.500000,9.000000,\Rx:=0.000000,\Ry:=0.000000),vel1,zoneval,Extruder\WObj:=Workobject_1;
MoveL RelTool (p1,5.000000,13.000000,9.000000,\Rx:=0.000000,\Ry:=-0.000000),vel1,zoneval,Extruder\WObj:=Workobject_1;
MoveL RelTool (p1,7.500000,13.000000,9.000000,\Rx:=0.000000,\Ry:=-0.000000),vel1,zoneval,Extruder\WObj:=Workobject_1;
MoveL RelTool (p1,10.000000,13.000000,9.000000,\Rx:=0.000000,\Ry:=-0.000000),vel1,zoneval,Extruder\WObj:=Workobject_1;
MoveL RelTool (p1,12.500000,13.000000,9.000000,\Rx:=0.000000,\Ry:=-0.000000),vel1,zoneval,Extruder\WObj:=Workobject_1;
MoveL RelTool (p1,15.000000,13.000000,9.000000,\Rx:=0.000000,\Ry:=-0.000000),vel1,zoneval,Extruder\WObj:=Workobject_1;
MoveL RelTool (p1,17.500000,13.000000,9.083964,\Rx:=0.000000,\Ry:=-4.411855),vel1,zoneval,Extruder\WObj:=Workobject_1;
MoveL RelTool (p1,20.000000,13.000000,11.367111,\Rx:=0.000000,\Ry:=-10.154539),vel1,zoneval,Extruder\WObj:=Workobject_1;
MoveL RelTool (p1,22.500000,13.000000,13.528177,\Rx:=0.000000,\Ry:=-7.985654),vel1,zoneval,Extruder\WObj:=Workobject_1;
MoveL RelTool (p1,25.000000,13.000000,15.076143,\Rx:=0.000000,\Ry:=-5.751524),vel1,zoneval,Extruder\WObj:=Workobject_1;
MoveL RelTool (p1,27.500000,13.000000,16.224522,\Rx:=0.000000,\Ry:=-4.442626),vel1,zoneval,Extruder\WObj:=Workobject_1;
MoveL RelTool (p1,30.000000,13.000000,17.115741,\Rx:=0.000000,\Ry:=-3.471339),vel1,zoneval,Extruder\WObj:=Workobject_1;
MoveL RelTool (p1,32.500000,13.000000,17.811501,\Rx:=0.000000,\Ry:=-2.537038),vel1,zoneval,Extruder\WObj:=Workobject_1;
MoveL RelTool (p1,35.000000,13.000000,18.316346,\Rx:=0.000000,\Ry:=-2.278631),vel1,zoneval,Extruder\WObj:=Workobject_1;
MoveL RelTool (p1,37.500000,13.000000,18.667838,\Rx:=0.000000,\Ry:=-1.652509),vel1,zoneval,Extruder\WObj:=Workobject_1;
MoveL RelTool (p1,40.000000,13.000000,18.885153,\Rx:=0.000000,\Ry:=-0.809967),vel1,zoneval,Extruder\WObj:=Workobject_1;
MoveL RelTool (p1,42.500000,13.000000,18.988071,\Rx:=0.000000,\Ry:=-0.131676),vel1,zoneval,Extruder\WObj:=Workobject_1;
MoveL RelTool (p1,45.000000,13.000000,18.928943,\Rx:=0.000000,\Ry:=0.547333),vel1,zoneval,Extruder\WObj:=Workobject_1;
MoveL RelTool (p1,47.500000,13.000000,18.755880,\Rx:=0.000000,\Ry:=1.375675),vel1,zoneval,Extruder\WObj:=Workobject_1;
MoveL RelTool (p1,50.000000,13.000000,18.449475,\Rx:=0.000000,\Ry:=2.217990),vel1,zoneval,Extruder\WObj:=Workobject_1;
MoveL RelTool (p1,52.500000,13.000000,17.996328,\Rx:=0.000000,\Ry:=3.108480),vel1,zoneval,Extruder\WObj:=Workobject_1;
MoveL RelTool (p1,55.000000,13.000000,17.373557,\Rx:=0.000000,\Ry:=4.006255),vel1,zoneval,Extruder\WObj:=Workobject_1;
MoveL RelTool (p1,57.500000,13.000000,16.553376,\Rx:=0.000000,\Ry:=5.005887),vel1,zoneval,Extruder\WObj:=Workobject_1;
MoveL RelTool (p1,60.000000,13.000000,15.484711,\Rx:=0.000000,\Ry:=6.061214),vel1,zoneval,Extruder\WObj:=Workobject_1;
MoveL RelTool (p1,62.500000,13.000000,14.090610,\Rx:=0.000000,\Ry:=7.227695),vel1,zoneval,Extruder\WObj:=Workobject_1;
MoveL RelTool (p1,65.000000,13.000000,12.198583,\Rx:=0.000000,\Ry:=9.902860),vel1,zoneval,Extruder\WObj:=Workobject_1;
MoveL RelTool (p1,67.500000,13.000000,9.464073,\Rx:=0.000000,\Ry:=6.326197),vel1,zoneval,Extruder\WObj:=Workobject_1;
MoveL RelTool (p1,70.000000,13.000000,9.000000,\Rx:=0.000000,\Ry:=-0.000000),vel1,zoneval,Extruder\WObj:=Workobject_1;
MoveL RelTool (p1,72.500000,13.000000,9.000000,\Rx:=0.000000,\Ry:=-0.000000),vel1,zoneval,Extruder\WObj:=Workobject_1;
MoveL RelTool (p1,75.000000,13.000000,9.000000,\Rx:=0.000000,\Ry:=-0.000000),vel1,zoneval,Extruder\WObj:=Workobject_1;
MoveL RelTool (p1,77.500000,13.000000,9.000000,\Rx:=0.000000,\Ry:=-0.000000),vel1,zoneval,Extruder\WObj:=Workobject_1;
MoveL RelTool (p1,80.000000,13.000000,9.000000,\Rx:=0.000000,\Ry:=-0.000000),vel1,zoneval,Extruder\WObj:=Workobject_1;
MoveL RelTool (p1,82.500000,13.000000,9.000000,\Rx:=0.000000,\Ry:=-0.000000),vel1,zoneval,Extruder\WObj:=Workobject_1;
MoveL RelTool (p1,80.500000,13.500000,9.000000,\Rx:=0.000000,\Ry:=0.000000),vel1,zoneval,Extruder\WObj:=Workobject_1;
MoveL RelTool (p1,78.000000,13.500000,9.000000,\Rx:=0.000000,\Ry:=0.000000),vel1,zoneval,Extruder\WObj:=Workobject_1;
MoveL RelTool (p1,75.500000,13.500000,9.000000,\Rx:=0.000000,\Ry:=0.000000),vel1,zoneval,Extruder\WObj:=Workobject_1;
MoveL RelTool (p1,73.000000,13.500000,9.000000,\Rx:=0.000000,\Ry:=0.000000),vel1,zoneval,Extruder\WObj:=Workobject_1;
MoveL RelTool (p1,70.500000,13.500000,9.000000,\Rx:=0.000000,\Ry:=0.000000),vel1,zoneval,Extruder\WObj:=Workobject_1;
MoveL RelTool (p1,68.000000,13.500000,9.192958,\Rx:=0.000000,\Ry:=6.326197),vel1,zoneval,Extruder\WObj:=Workobject_1;
MoveL RelTool (p1,65.500000,13.500000,11.706154,\Rx:=0.000000,\Ry:=9.902860),vel1,zoneval,Extruder\WObj:=Workobject_1;
MoveL RelTool (p1,63.000000,13.500000,13.771773,\Rx:=0.000000,\Ry:=7.227695),vel1,zoneval,Extruder\WObj:=Workobject_1;
MoveL RelTool (p1,60.500000,13.500000,15.226913,\Rx:=0.000000,\Ry:=6.061214),vel1,zoneval,Extruder\WObj:=Workobject_1;
MoveL RelTool (p1,58.000000,13.500000,16.345998,\Rx:=0.000000,\Ry:=5.005887),vel1,zoneval,Extruder\WObj:=Workobject_1;
MoveL RelTool (p1,55.500000,13.500000,17.210825,\Rx:=0.000000,\Ry:=4.006255),vel1,zoneval,Extruder\WObj:=Workobject_1;
MoveL RelTool (p1,53.000000,13.500000,17.871774,\Rx:=0.000000,\Ry:=3.108480),vel1,zoneval,Extruder\WObj:=Workobject_1;
MoveL RelTool (p1,50.500000,13.500000,18.361483,\Rx:=0.000000,\Ry:=2.217990),vel1,zoneval,Extruder\WObj:=Workobject_1;
MoveL RelTool (p1,48.000000,13.500000,18.701647,\Rx:=0.000000,\Ry:=1.375675),vel1,zoneval,Extruder\WObj:=Workobject_1;
MoveL RelTool (p1,45.500000,13.500000,18.907436,\Rx:=0.000000,\Ry:=0.547333),vel1,zoneval,Extruder\WObj:=Workobject_1;
MoveL RelTool (p1,43.000000,13.500000,18.993242,\Rx:=0.000000,\Ry:=-0.131676),vel1,zoneval,Extruder\WObj:=Workobject_1;
MoveL RelTool (p1,40.500000,13.500000,18.917003,\Rx:=0.000000,\Ry:=-0.809967),vel1,zoneval,Extruder\WObj:=Workobject_1;
MoveL RelTool (p1,38.000000,13.500000,18.733099,\Rx:=0.000000,\Ry:=-1.652509),vel1,zoneval,Extruder\WObj:=Workobject_1;
MoveL RelTool (p1,35.500000,13.500000,18.406795,\Rx:=0.000000,\Ry:=-2.278631),vel1,zoneval,Extruder\WObj:=Workobject_1;
MoveL RelTool (p1,33.000000,13.500000,17.912470,\Rx:=0.000000,\Ry:=-2.537038),vel1,zoneval,Extruder\WObj:=Workobject_1;
MoveL RelTool (p1,30.500000,13.500000,17.255542,\Rx:=0.000000,\Ry:=-3.471339),vel1,zoneval,Extruder\WObj:=Workobject_1;
MoveL RelTool (p1,28.000000,13.500000,16.406426,\Rx:=0.000000,\Ry:=-4.442626),vel1,zoneval,Extruder\WObj:=Workobject_1;
MoveL RelTool (p1,25.500000,13.500000,15.318735,\Rx:=0.000000,\Ry:=-5.751524),vel1,zoneval,Extruder\WObj:=Workobject_1;
MoveL RelTool (p1,23.000000,13.500000,13.890588,\Rx:=0.000000,\Ry:=-7.985654),vel1,zoneval,Extruder\WObj:=Workobject_1;
MoveL RelTool (p1,20.500000,13.500000,11.879398,\Rx:=0.000000,\Ry:=-10.154539),vel1,zoneval,Extruder\WObj:=Workobject_1;
MoveL RelTool (p1,18.000000,13.500000,9.264501,\Rx:=0.000000,\Ry:=-4.411855),vel1,zoneval,Extruder\WObj:=Workobject_1;
MoveL RelTool (p1,15.500000,13.500000,9.000000,\Rx:=0.000000,\Ry:=0.000000),vel1,zoneval,Extruder\WObj:=Workobject_1;
MoveL RelTool (p1,13.000000,13.500000,9.000000,\Rx:=0.000000,\Ry:=0.000000),vel1,zoneval,Extruder\WObj:=Workobject_1;
MoveL RelTool (p1,10.500000,13.500000,9.000000,\Rx:=0.000000,\Ry:=0.000000),vel1,zoneval,Extruder\WObj:=Workobject_1;
MoveL RelTool (p1,8.000000,13.500000,9.000000,\Rx:=0.000000,\Ry:=0.000000),vel1,zoneval,Extruder\WObj:=Workobject_1;
MoveL RelTool (p1,5.500000,13.500000,9.000000,\Rx:=0.000000,\Ry:=0.000000),vel1,zoneval,Extruder\WObj:=Workobject_1;
MoveL RelTool (p1,3.000000,13.500000,9.000000,\Rx:=0.000000,\Ry:=0.000000),vel1,zoneval,Extruder\WObj:=Workobject_1;
MoveL RelTool (p1,5.000000,14.000000,9.000000,\Rx:=0.000000,\Ry:=-0.000000),vel1,zoneval,Extruder\WObj:=Workobject_1;
MoveL RelTool (p1,7.500000,14.000000,9.000000,\Rx:=0.000000,\Ry:=-0.000000),vel1,zoneval,Extruder\WObj:=Workobject_1;
MoveL RelTool (p1,10.000000,14.000000,9.000000,\Rx:=0.000000,\Ry:=-0.000000),vel1,zoneval,Extruder\WObj:=Workobject_1;
MoveL RelTool (p1,12.500000,14.000000,9.000000,\Rx:=0.000000,\Ry:=-0.000000),vel1,zoneval,Extruder\WObj:=Workobject_1;
MoveL RelTool (p1,15.000000,14.000000,9.000000,\Rx:=0.000000,\Ry:=-0.000000),vel1,zoneval,Extruder\WObj:=Workobject_1;
MoveL RelTool (p1,17.500000,14.000000,9.083964,\Rx:=0.000000,\Ry:=-4.411855),vel1,zoneval,Extruder\WObj:=Workobject_1;
MoveL RelTool (p1,20.000000,14.000000,11.367111,\Rx:=0.000000,\Ry:=-10.154539),vel1,zoneval,Extruder\WObj:=Workobject_1;
MoveL RelTool (p1,22.500000,14.000000,13.528177,\Rx:=0.000000,\Ry:=-7.985654),vel1,zoneval,Extruder\WObj:=Workobject_1;
MoveL RelTool (p1,25.000000,14.000000,15.076143,\Rx:=0.000000,\Ry:=-5.751524),vel1,zoneval,Extruder\WObj:=Workobject_1;
MoveL RelTool (p1,27.500000,14.000000,16.224522,\Rx:=0.000000,\Ry:=-4.442626),vel1,zoneval,Extruder\WObj:=Workobject_1;
MoveL RelTool (p1,30.000000,14.000000,17.115741,\Rx:=0.000000,\Ry:=-3.471339),vel1,zoneval,Extruder\WObj:=Workobject_1;
MoveL RelTool (p1,32.500000,14.000000,17.811501,\Rx:=0.000000,\Ry:=-2.537038),vel1,zoneval,Extruder\WObj:=Workobject_1;
MoveL RelTool (p1,35.000000,14.000000,18.316346,\Rx:=0.000000,\Ry:=-2.278631),vel1,zoneval,Extruder\WObj:=Workobject_1;
MoveL RelTool (p1,37.500000,14.000000,18.667838,\Rx:=0.000000,\Ry:=-1.652509),vel1,zoneval,Extruder\WObj:=Workobject_1;
MoveL RelTool (p1,40.000000,14.000000,18.885153,\Rx:=0.000000,\Ry:=-0.809967),vel1,zoneval,Extruder\WObj:=Workobject_1;
MoveL RelTool (p1,42.500000,14.000000,18.988071,\Rx:=0.000000,\Ry:=-0.131676),vel1,zoneval,Extruder\WObj:=Workobject_1;
MoveL RelTool (p1,45.000000,14.000000,18.928943,\Rx:=0.000000,\Ry:=0.547333),vel1,zoneval,Extruder\WObj:=Workobject_1;
MoveL RelTool (p1,47.500000,14.000000,18.755880,\Rx:=0.000000,\Ry:=1.375675),vel1,zoneval,Extruder\WObj:=Workobject_1;
MoveL RelTool (p1,50.000000,14.000000,18.449475,\Rx:=0.000000,\Ry:=2.217990),vel1,zoneval,Extruder\WObj:=Workobject_1;
MoveL RelTool (p1,52.500000,14.000000,17.996328,\Rx:=0.000000,\Ry:=3.108480),vel1,zoneval,Extruder\WObj:=Workobject_1;
MoveL RelTool (p1,55.000000,14.000000,17.373557,\Rx:=0.000000,\Ry:=4.006255),vel1,zoneval,Extruder\WObj:=Workobject_1;
MoveL RelTool (p1,57.500000,14.000000,16.553376,\Rx:=0.000000,\Ry:=5.005887),vel1,zoneval,Extruder\WObj:=Workobject_1;
MoveL RelTool (p1,60.000000,14.000000,15.484711,\Rx:=0.000000,\Ry:=6.061214),vel1,zoneval,Extruder\WObj:=Workobject_1;
MoveL RelTool (p1,62.500000,14.000000,14.090610,\Rx:=0.000000,\Ry:=7.227695),vel1,zoneval,Extruder\WObj:=Workobject_1;
MoveL RelTool (p1,65.000000,14.000000,12.198583,\Rx:=0.000000,\Ry:=9.902860),vel1,zoneval,Extruder\WObj:=Workobject_1;
MoveL RelTool (p1,67.500000,14.000000,9.464073,\Rx:=0.000000,\Ry:=6.326197),vel1,zoneval,Extruder\WObj:=Workobject_1;
MoveL RelTool (p1,70.000000,14.000000,9.000000,\Rx:=0.000000,\Ry:=-0.000000),vel1,zoneval,Extruder\WObj:=Workobject_1;
MoveL RelTool (p1,72.500000,14.000000,9.000000,\Rx:=0.000000,\Ry:=-0.000000),vel1,zoneval,Extruder\WObj:=Workobject_1;
MoveL RelTool (p1,75.000000,14.000000,9.000000,\Rx:=0.000000,\Ry:=-0.000000),vel1,zoneval,Extruder\WObj:=Workobject_1;
MoveL RelTool (p1,77.500000,14.000000,9.000000,\Rx:=0.000000,\Ry:=-0.000000),vel1,zoneval,Extruder\WObj:=Workobject_1;
MoveL RelTool (p1,80.000000,14.000000,9.000000,\Rx:=0.000000,\Ry:=-0.000000),vel1,zoneval,Extruder\WObj:=Workobject_1;
MoveL RelTool (p1,82.500000,14.000000,9.000000,\Rx:=0.000000,\Ry:=-0.000000),vel1,zoneval,Extruder\WObj:=Workobject_1;
MoveL RelTool (p1,80.500000,14.500000,9.000000,\Rx:=0.000000,\Ry:=0.000000),vel1,zoneval,Extruder\WObj:=Workobject_1;
MoveL RelTool (p1,78.000000,14.500000,9.000000,\Rx:=0.000000,\Ry:=0.000000),vel1,zoneval,Extruder\WObj:=Workobject_1;
MoveL RelTool (p1,75.500000,14.500000,9.000000,\Rx:=0.000000,\Ry:=0.000000),vel1,zoneval,Extruder\WObj:=Workobject_1;
MoveL RelTool (p1,73.000000,14.500000,9.000000,\Rx:=0.000000,\Ry:=0.000000),vel1,zoneval,Extruder\WObj:=Workobject_1;
MoveL RelTool (p1,70.500000,14.500000,9.000000,\Rx:=0.000000,\Ry:=0.000000),vel1,zoneval,Extruder\WObj:=Workobject_1;
MoveL RelTool (p1,68.000000,14.500000,9.192958,\Rx:=0.000000,\Ry:=6.326197),vel1,zoneval,Extruder\WObj:=Workobject_1;
MoveL RelTool (p1,65.500000,14.500000,11.706154,\Rx:=0.000000,\Ry:=9.902860),vel1,zoneval,Extruder\WObj:=Workobject_1;
MoveL RelTool (p1,63.000000,14.500000,13.771773,\Rx:=0.000000,\Ry:=7.227695),vel1,zoneval,Extruder\WObj:=Workobject_1;
MoveL RelTool (p1,60.500000,14.500000,15.226913,\Rx:=0.000000,\Ry:=6.061214),vel1,zoneval,Extruder\WObj:=Workobject_1;
MoveL RelTool (p1,58.000000,14.500000,16.345998,\Rx:=0.000000,\Ry:=5.005887),vel1,zoneval,Extruder\WObj:=Workobject_1;
MoveL RelTool (p1,55.500000,14.500000,17.210825,\Rx:=0.000000,\Ry:=4.006255),vel1,zoneval,Extruder\WObj:=Workobject_1;
MoveL RelTool (p1,53.000000,14.500000,17.871774,\Rx:=0.000000,\Ry:=3.108480),vel1,zoneval,Extruder\WObj:=Workobject_1;
MoveL RelTool (p1,50.500000,14.500000,18.361483,\Rx:=0.000000,\Ry:=2.217990),vel1,zoneval,Extruder\WObj:=Workobject_1;
MoveL RelTool (p1,48.000000,14.500000,18.701647,\Rx:=0.000000,\Ry:=1.375675),vel1,zoneval,Extruder\WObj:=Workobject_1;
MoveL RelTool (p1,45.500000,14.500000,18.907436,\Rx:=0.000000,\Ry:=0.547333),vel1,zoneval,Extruder\WObj:=Workobject_1;
MoveL RelTool (p1,43.000000,14.500000,18.993242,\Rx:=0.000000,\Ry:=-0.131676),vel1,zoneval,Extruder\WObj:=Workobject_1;
MoveL RelTool (p1,40.500000,14.500000,18.917003,\Rx:=0.000000,\Ry:=-0.809967),vel1,zoneval,Extruder\WObj:=Workobject_1;
MoveL RelTool (p1,38.000000,14.500000,18.733099,\Rx:=0.000000,\Ry:=-1.652509),vel1,zoneval,Extruder\WObj:=Workobject_1;
MoveL RelTool (p1,35.500000,14.500000,18.406795,\Rx:=0.000000,\Ry:=-2.278631),vel1,zoneval,Extruder\WObj:=Workobject_1;
MoveL RelTool (p1,33.000000,14.500000,17.912470,\Rx:=0.000000,\Ry:=-2.537038),vel1,zoneval,Extruder\WObj:=Workobject_1;
MoveL RelTool (p1,30.500000,14.500000,17.255542,\Rx:=0.000000,\Ry:=-3.471339),vel1,zoneval,Extruder\WObj:=Workobject_1;
MoveL RelTool (p1,28.000000,14.500000,16.406426,\Rx:=0.000000,\Ry:=-4.442626),vel1,zoneval,Extruder\WObj:=Workobject_1;
MoveL RelTool (p1,25.500000,14.500000,15.318735,\Rx:=0.000000,\Ry:=-5.751524),vel1,zoneval,Extruder\WObj:=Workobject_1;
MoveL RelTool (p1,23.000000,14.500000,13.890588,\Rx:=0.000000,\Ry:=-7.985654),vel1,zoneval,Extruder\WObj:=Workobject_1;
MoveL RelTool (p1,20.500000,14.500000,11.879398,\Rx:=0.000000,\Ry:=-10.154539),vel1,zoneval,Extruder\WObj:=Workobject_1;
MoveL RelTool (p1,18.000000,14.500000,9.264501,\Rx:=0.000000,\Ry:=-4.411855),vel1,zoneval,Extruder\WObj:=Workobject_1;
MoveL RelTool (p1,15.500000,14.500000,9.000000,\Rx:=0.000000,\Ry:=0.000000),vel1,zoneval,Extruder\WObj:=Workobject_1;
MoveL RelTool (p1,13.000000,14.500000,9.000000,\Rx:=0.000000,\Ry:=0.000000),vel1,zoneval,Extruder\WObj:=Workobject_1;
MoveL RelTool (p1,10.500000,14.500000,9.000000,\Rx:=0.000000,\Ry:=0.000000),vel1,zoneval,Extruder\WObj:=Workobject_1;
MoveL RelTool (p1,8.000000,14.500000,9.000000,\Rx:=0.000000,\Ry:=0.000000),vel1,zoneval,Extruder\WObj:=Workobject_1;
MoveL RelTool (p1,5.500000,14.500000,9.000000,\Rx:=0.000000,\Ry:=0.000000),vel1,zoneval,Extruder\WObj:=Workobject_1;
MoveL RelTool (p1,3.000000,14.500000,9.000000,\Rx:=0.000000,\Ry:=0.000000),vel1,zoneval,Extruder\WObj:=Workobject_1;
MoveL RelTool (p1,5.000000,15.000000,9.000000,\Rx:=0.000000,\Ry:=-0.000000),vel1,zoneval,Extruder\WObj:=Workobject_1;
MoveL RelTool (p1,7.500000,15.000000,9.000000,\Rx:=0.000000,\Ry:=-0.000000),vel1,zoneval,Extruder\WObj:=Workobject_1;
MoveL RelTool (p1,10.000000,15.000000,9.000000,\Rx:=0.000000,\Ry:=-0.000000),vel1,zoneval,Extruder\WObj:=Workobject_1;
MoveL RelTool (p1,12.500000,15.000000,9.000000,\Rx:=0.000000,\Ry:=-0.000000),vel1,zoneval,Extruder\WObj:=Workobject_1;
MoveL RelTool (p1,15.000000,15.000000,9.000000,\Rx:=0.000000,\Ry:=-0.000000),vel1,zoneval,Extruder\WObj:=Workobject_1;
MoveL RelTool (p1,17.500000,15.000000,9.083964,\Rx:=0.000000,\Ry:=-4.411855),vel1,zoneval,Extruder\WObj:=Workobject_1;
MoveL RelTool (p1,20.000000,15.000000,11.367111,\Rx:=0.000000,\Ry:=-10.154539),vel1,zoneval,Extruder\WObj:=Workobject_1;
MoveL RelTool (p1,22.500000,15.000000,13.528177,\Rx:=0.000000,\Ry:=-7.985654),vel1,zoneval,Extruder\WObj:=Workobject_1;
MoveL RelTool (p1,25.000000,15.000000,15.076143,\Rx:=0.000000,\Ry:=-5.751524),vel1,zoneval,Extruder\WObj:=Workobject_1;
MoveL RelTool (p1,27.500000,15.000000,16.224522,\Rx:=0.000000,\Ry:=-4.442626),vel1,zoneval,Extruder\WObj:=Workobject_1;
MoveL RelTool (p1,30.000000,15.000000,17.115741,\Rx:=0.000000,\Ry:=-3.471339),vel1,zoneval,Extruder\WObj:=Workobject_1;
MoveL RelTool (p1,32.500000,15.000000,17.811501,\Rx:=0.000000,\Ry:=-2.537038),vel1,zoneval,Extruder\WObj:=Workobject_1;
MoveL RelTool (p1,35.000000,15.000000,18.316346,\Rx:=0.000000,\Ry:=-2.278631),vel1,zoneval,Extruder\WObj:=Workobject_1;
MoveL RelTool (p1,37.500000,15.000000,18.667838,\Rx:=0.000000,\Ry:=-1.652509),vel1,zoneval,Extruder\WObj:=Workobject_1;
MoveL RelTool (p1,40.000000,15.000000,18.885153,\Rx:=0.000000,\Ry:=-0.809967),vel1,zoneval,Extruder\WObj:=Workobject_1;
MoveL RelTool (p1,42.500000,15.000000,18.988071,\Rx:=0.000000,\Ry:=-0.131676),vel1,zoneval,Extruder\WObj:=Workobject_1;
MoveL RelTool (p1,45.000000,15.000000,18.928943,\Rx:=0.000000,\Ry:=0.547333),vel1,zoneval,Extruder\WObj:=Workobject_1;
MoveL RelTool (p1,47.500000,15.000000,18.755880,\Rx:=0.000000,\Ry:=1.375675),vel1,zoneval,Extruder\WObj:=Workobject_1;
MoveL RelTool (p1,50.000000,15.000000,18.449475,\Rx:=0.000000,\Ry:=2.217990),vel1,zoneval,Extruder\WObj:=Workobject_1;
MoveL RelTool (p1,52.500000,15.000000,17.996328,\Rx:=0.000000,\Ry:=3.108480),vel1,zoneval,Extruder\WObj:=Workobject_1;
MoveL RelTool (p1,55.000000,15.000000,17.373557,\Rx:=0.000000,\Ry:=4.006255),vel1,zoneval,Extruder\WObj:=Workobject_1;
MoveL RelTool (p1,57.500000,15.000000,16.553376,\Rx:=0.000000,\Ry:=5.005887),vel1,zoneval,Extruder\WObj:=Workobject_1;
MoveL RelTool (p1,60.000000,15.000000,15.484711,\Rx:=0.000000,\Ry:=6.061214),vel1,zoneval,Extruder\WObj:=Workobject_1;
MoveL RelTool (p1,62.500000,15.000000,14.090610,\Rx:=0.000000,\Ry:=7.227695),vel1,zoneval,Extruder\WObj:=Workobject_1;
MoveL RelTool (p1,65.000000,15.000000,12.198583,\Rx:=0.000000,\Ry:=9.902860),vel1,zoneval,Extruder\WObj:=Workobject_1;
MoveL RelTool (p1,67.500000,15.000000,9.464073,\Rx:=0.000000,\Ry:=6.326197),vel1,zoneval,Extruder\WObj:=Workobject_1;
MoveL RelTool (p1,70.000000,15.000000,9.000000,\Rx:=0.000000,\Ry:=-0.000000),vel1,zoneval,Extruder\WObj:=Workobject_1;
MoveL RelTool (p1,72.500000,15.000000,9.000000,\Rx:=0.000000,\Ry:=-0.000000),vel1,zoneval,Extruder\WObj:=Workobject_1;
MoveL RelTool (p1,75.000000,15.000000,9.000000,\Rx:=0.000000,\Ry:=-0.000000),vel1,zoneval,Extruder\WObj:=Workobject_1;
MoveL RelTool (p1,77.500000,15.000000,9.000000,\Rx:=0.000000,\Ry:=-0.000000),vel1,zoneval,Extruder\WObj:=Workobject_1;
MoveL RelTool (p1,80.000000,15.000000,9.000000,\Rx:=0.000000,\Ry:=-0.000000),vel1,zoneval,Extruder\WObj:=Workobject_1;
MoveL RelTool (p1,82.500000,15.000000,9.000000,\Rx:=0.000000,\Ry:=-0.000000),vel1,zoneval,Extruder\WObj:=Workobject_1;
MoveL RelTool (p1,80.500000,15.500000,9.000000,\Rx:=0.000000,\Ry:=0.000000),vel1,zoneval,Extruder\WObj:=Workobject_1;
MoveL RelTool (p1,78.000000,15.500000,9.000000,\Rx:=0.000000,\Ry:=0.000000),vel1,zoneval,Extruder\WObj:=Workobject_1;
MoveL RelTool (p1,75.500000,15.500000,9.000000,\Rx:=0.000000,\Ry:=0.000000),vel1,zoneval,Extruder\WObj:=Workobject_1;
MoveL RelTool (p1,73.000000,15.500000,9.000000,\Rx:=0.000000,\Ry:=0.000000),vel1,zoneval,Extruder\WObj:=Workobject_1;
MoveL RelTool (p1,70.500000,15.500000,9.000000,\Rx:=0.000000,\Ry:=0.000000),vel1,zoneval,Extruder\WObj:=Workobject_1;
MoveL RelTool (p1,68.000000,15.500000,9.192958,\Rx:=0.000000,\Ry:=6.326197),vel1,zoneval,Extruder\WObj:=Workobject_1;
MoveL RelTool (p1,65.500000,15.500000,11.706154,\Rx:=0.000000,\Ry:=9.902860),vel1,zoneval,Extruder\WObj:=Workobject_1;
MoveL RelTool (p1,63.000000,15.500000,13.771773,\Rx:=0.000000,\Ry:=7.227695),vel1,zoneval,Extruder\WObj:=Workobject_1;
MoveL RelTool (p1,60.500000,15.500000,15.226913,\Rx:=0.000000,\Ry:=6.061214),vel1,zoneval,Extruder\WObj:=Workobject_1;
MoveL RelTool (p1,58.000000,15.500000,16.345998,\Rx:=0.000000,\Ry:=5.005887),vel1,zoneval,Extruder\WObj:=Workobject_1;
MoveL RelTool (p1,55.500000,15.500000,17.210825,\Rx:=0.000000,\Ry:=4.006255),vel1,zoneval,Extruder\WObj:=Workobject_1;
MoveL RelTool (p1,53.000000,15.500000,17.871774,\Rx:=0.000000,\Ry:=3.108480),vel1,zoneval,Extruder\WObj:=Workobject_1;
MoveL RelTool (p1,50.500000,15.500000,18.361483,\Rx:=0.000000,\Ry:=2.217990),vel1,zoneval,Extruder\WObj:=Workobject_1;
MoveL RelTool (p1,48.000000,15.500000,18.701647,\Rx:=0.000000,\Ry:=1.375675),vel1,zoneval,Extruder\WObj:=Workobject_1;
MoveL RelTool (p1,45.500000,15.500000,18.907436,\Rx:=0.000000,\Ry:=0.547333),vel1,zoneval,Extruder\WObj:=Workobject_1;
MoveL RelTool (p1,43.000000,15.500000,18.993242,\Rx:=0.000000,\Ry:=-0.131676),vel1,zoneval,Extruder\WObj:=Workobject_1;
MoveL RelTool (p1,40.500000,15.500000,18.917003,\Rx:=0.000000,\Ry:=-0.809967),vel1,zoneval,Extruder\WObj:=Workobject_1;
MoveL RelTool (p1,38.000000,15.500000,18.733099,\Rx:=0.000000,\Ry:=-1.652509),vel1,zoneval,Extruder\WObj:=Workobject_1;
MoveL RelTool (p1,35.500000,15.500000,18.406795,\Rx:=0.000000,\Ry:=-2.278631),vel1,zoneval,Extruder\WObj:=Workobject_1;
MoveL RelTool (p1,33.000000,15.500000,17.912470,\Rx:=0.000000,\Ry:=-2.537038),vel1,zoneval,Extruder\WObj:=Workobject_1;
MoveL RelTool (p1,30.500000,15.500000,17.255542,\Rx:=0.000000,\Ry:=-3.471339),vel1,zoneval,Extruder\WObj:=Workobject_1;
MoveL RelTool (p1,28.000000,15.500000,16.406426,\Rx:=0.000000,\Ry:=-4.442626),vel1,zoneval,Extruder\WObj:=Workobject_1;
MoveL RelTool (p1,25.500000,15.500000,15.318735,\Rx:=0.000000,\Ry:=-5.751524),vel1,zoneval,Extruder\WObj:=Workobject_1;
MoveL RelTool (p1,23.000000,15.500000,13.890588,\Rx:=0.000000,\Ry:=-7.985654),vel1,zoneval,Extruder\WObj:=Workobject_1;
MoveL RelTool (p1,20.500000,15.500000,11.879398,\Rx:=0.000000,\Ry:=-10.154539),vel1,zoneval,Extruder\WObj:=Workobject_1;
MoveL RelTool (p1,18.000000,15.500000,9.264501,\Rx:=0.000000,\Ry:=-4.411855),vel1,zoneval,Extruder\WObj:=Workobject_1;
MoveL RelTool (p1,15.500000,15.500000,9.000000,\Rx:=0.000000,\Ry:=0.000000),vel1,zoneval,Extruder\WObj:=Workobject_1;
MoveL RelTool (p1,13.000000,15.500000,9.000000,\Rx:=0.000000,\Ry:=0.000000),vel1,zoneval,Extruder\WObj:=Workobject_1;
MoveL RelTool (p1,10.500000,15.500000,9.000000,\Rx:=0.000000,\Ry:=0.000000),vel1,zoneval,Extruder\WObj:=Workobject_1;
MoveL RelTool (p1,8.000000,15.500000,9.000000,\Rx:=0.000000,\Ry:=0.000000),vel1,zoneval,Extruder\WObj:=Workobject_1;
MoveL RelTool (p1,5.500000,15.500000,9.000000,\Rx:=0.000000,\Ry:=0.000000),vel1,zoneval,Extruder\WObj:=Workobject_1;
MoveL RelTool (p1,3.000000,15.500000,9.000000,\Rx:=0.000000,\Ry:=0.000000),vel1,zoneval,Extruder\WObj:=Workobject_1;
MoveL RelTool (p1,5.000000,16.000000,9.000000,\Rx:=0.000000,\Ry:=-0.000000),vel1,zoneval,Extruder\WObj:=Workobject_1;
MoveL RelTool (p1,7.500000,16.000000,9.000000,\Rx:=0.000000,\Ry:=-0.000000),vel1,zoneval,Extruder\WObj:=Workobject_1;
MoveL RelTool (p1,10.000000,16.000000,9.000000,\Rx:=0.000000,\Ry:=-0.000000),vel1,zoneval,Extruder\WObj:=Workobject_1;
MoveL RelTool (p1,12.500000,16.000000,9.000000,\Rx:=0.000000,\Ry:=-0.000000),vel1,zoneval,Extruder\WObj:=Workobject_1;
MoveL RelTool (p1,15.000000,16.000000,9.000000,\Rx:=0.000000,\Ry:=-0.000000),vel1,zoneval,Extruder\WObj:=Workobject_1;
MoveL RelTool (p1,17.500000,16.000000,9.083964,\Rx:=0.000000,\Ry:=-4.411855),vel1,zoneval,Extruder\WObj:=Workobject_1;
MoveL RelTool (p1,20.000000,16.000000,11.367111,\Rx:=0.000000,\Ry:=-10.154539),vel1,zoneval,Extruder\WObj:=Workobject_1;
MoveL RelTool (p1,22.500000,16.000000,13.528177,\Rx:=0.000000,\Ry:=-7.985654),vel1,zoneval,Extruder\WObj:=Workobject_1;
MoveL RelTool (p1,25.000000,16.000000,15.076143,\Rx:=0.000000,\Ry:=-5.751524),vel1,zoneval,Extruder\WObj:=Workobject_1;
MoveL RelTool (p1,27.500000,16.000000,16.224522,\Rx:=0.000000,\Ry:=-4.442626),vel1,zoneval,Extruder\WObj:=Workobject_1;
